// NETWORK 2
// (* End of system generated code, could be modified for your application *)
xExitStop := xCMDwasActive AND NOT stMachineInterface.q_xCmdActive OR xReactionActive;
END_ACTION

ACTION AutoStop_Entry:
(* System generated code, could be modified for your application *)
	xCMDwasActive:=FALSE;
	IF	xReactionActive	THEN
		;
	ELSIF stMachineInterface.q_xCmdDone AND NOT stMachineInterface.q_xCmdActive THEN
		stMachineInterface.iq_diCmd := ET_Cmd.StopAuto;
	ELSE
		stMachineInterface.iq_diCmd := ET_Cmd.Abort;
	END_IF
(* End of system generated code, could be modified for your application *)
END_ACTION

ACTION InitModule_Action:
(* This step is used for initialisations after being enabled *)

(* System generated code, do not change without consulting 'Schneider Electric Automation GmbH' - otherwise you risk instability!!!*)


stMachineInterface.q_xActive		:= TRUE;
stMachineInterface.q_xReady			:= FALSE;
stMachineInterface.q_etDiag			:= GD.ET_Diag.Ok;
stMachineInterface.q_udiDiagExt		:= ET_DiagExt.Initializing;
stMachineInterface.q_sDiagExt		:= FC_EtDiagExtToString(ET_DiagExt.Initializing);
stMachineInterface.q_sMsg			:= '';

stMachineInterface.i_sModuleName		:= 'MainMachine';
stMachineInterface.i_udiModuleId		:= c_udiMainModuleId;
stMachineInterface.i_xLogEnable			:= TRUE;
stMachineInterface.i_wLogDataFilter		:= UDINT_TO_WORD(TPL.ET_LogDataFilter.ModuleDefault);

fbLoggerPoint.RegisterLoggerPoint(	i_ifParent		:= APL.G_ifApplicationLogger,
									i_sName			:= stMachineInterface.i_sModuleName,
									i_sType			:= 'MainMachine',
									i_sSource		:= 'Project',
									q_etDiag		=> ,
									q_etDiagExt		=> );
fbModuleController.RegisterLoggerPoint(	i_ifParent	:= fbLoggerPoint,
										i_sName		:= 'ModuleController',
										q_etDiag	=> ,
										q_etDiagExt	=> );
fbExceptionHandler.RegisterLoggerPoint(	i_ifParent	:= fbLoggerPoint,
										i_sName		:= 'ExceptionHandler',
										q_etDiag	=> ,
										q_etDiagExt	=> );

SYSTEMINTERFACE.FC_DiagNoQuitSet(i_diDiagCode := 8316);
SYSTEMINTERFACE.FC_DiagConfigSet(i_diDiagCode := 8252,i_diDiagClass := 1);
(* End of system generated code, do not change without consulting 'Schneider Electric Automation GmbH' - otherwise you risk instability!!!*)

(* System generated code, could be modified for your application *)
Init_Exceptions();
(* End of system generated code, could be modified for your application *)

(* System generated code, do not change without consulting 'Schneider Electric Automation GmbH' - otherwise you risk instability!!!*)
Init_SubModules();
Init_CmdTables();
Init_Reactions();
UpdateStructs();
(* End of system generated code, do not change without consulting 'Schneider Electric Automation GmbH' - otherwise you risk instability!!!*)

(* System generated code, could be modified for your application *)
Init_Alpha();
Init_Bravo();
Init_MultiCarrier();

xInitSuccessful := TRUE;

(* End of system generated code, could be modified for your application *)

(* Application specific code *)
(* ToDo: Add your application specific code here *)
;
(* End of application specific code *)
END_ACTION

ACTION Input_Action:
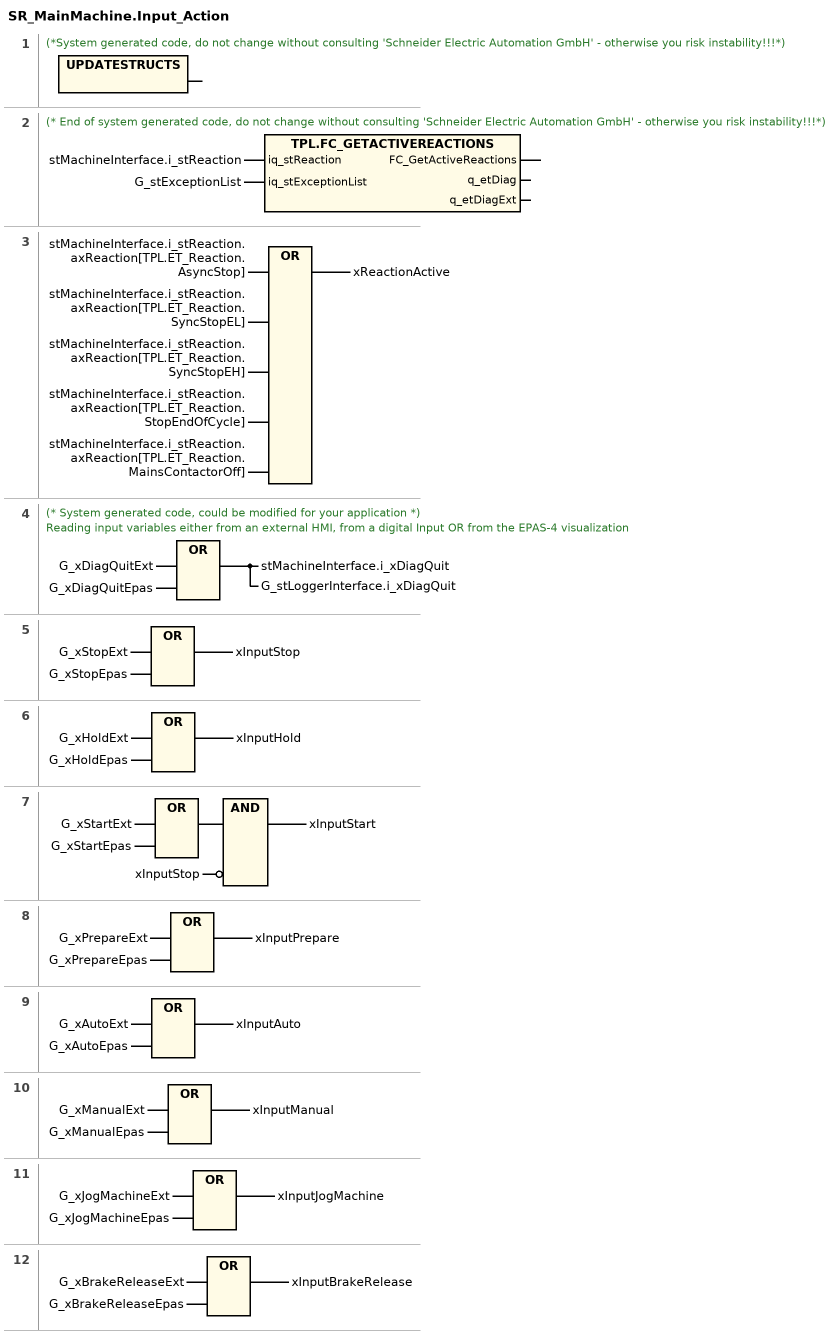
// NETWORK 1
// (*System generated code, do not change without consulting 'Schneider Electric Automation GmbH' - otherwise you risk instability!!!*)
UPDATESTRUCTS();

// NETWORK 2
// (* End of system generated code, do not change without consulting 'Schneider Electric Automation GmbH' - otherwise you risk instability!!!*)
TPL.FC_GETACTIVEREACTIONS(iq_stReaction := stMachineInterface.i_stReaction, iq_stExceptionList := G_stExceptionList);

// NETWORK 3
xReactionActive := stMachineInterface.i_stReaction.axReaction[TPL.ET_Reaction.AsyncStop] OR stMachineInterface.i_stReaction.axReaction[TPL.ET_Reaction.SyncStopEL] OR stMachineInterface.i_stReaction.axReaction[TPL.ET_Reaction.SyncStopEH] OR stMachineInterface.i_stReaction.axReaction[TPL.ET_Reaction.StopEndOfCycle] OR stMachineInterface.i_stReaction.axReaction[TPL.ET_Reaction.MainsContactorOff];

// NETWORK 4
// 					(* System generated code, could be modified for your application *)
// Reading input variables either from an external HMI, from a digital Input OR from the EPAS-4 visualization
//
_w1 := G_xDiagQuitExt OR G_xDiagQuitEpas;
stMachineInterface.i_xDiagQuit := _w1;
G_stLoggerInterface.i_xDiagQuit := _w1;

// NETWORK 5
xInputStop := G_xStopExt OR G_xStopEpas;

// NETWORK 6
xInputHold := G_xHoldExt OR G_xHoldEpas;

// NETWORK 7
xInputStart := (G_xStartExt OR G_xStartEpas) AND NOT xInputStop;

// NETWORK 8
xInputPrepare := G_xPrepareExt OR G_xPrepareEpas;

// NETWORK 9
xInputAuto := G_xAutoExt OR G_xAutoEpas;

// NETWORK 10
xInputManual := G_xManualExt OR G_xManualEpas;

// NETWORK 11
xInputJogMachine := G_xJogMachineExt OR G_xJogMachineEpas;

// NETWORK 12
xInputBrakeRelease := G_xBrakeReleaseExt OR G_xBrakeReleaseEpas;

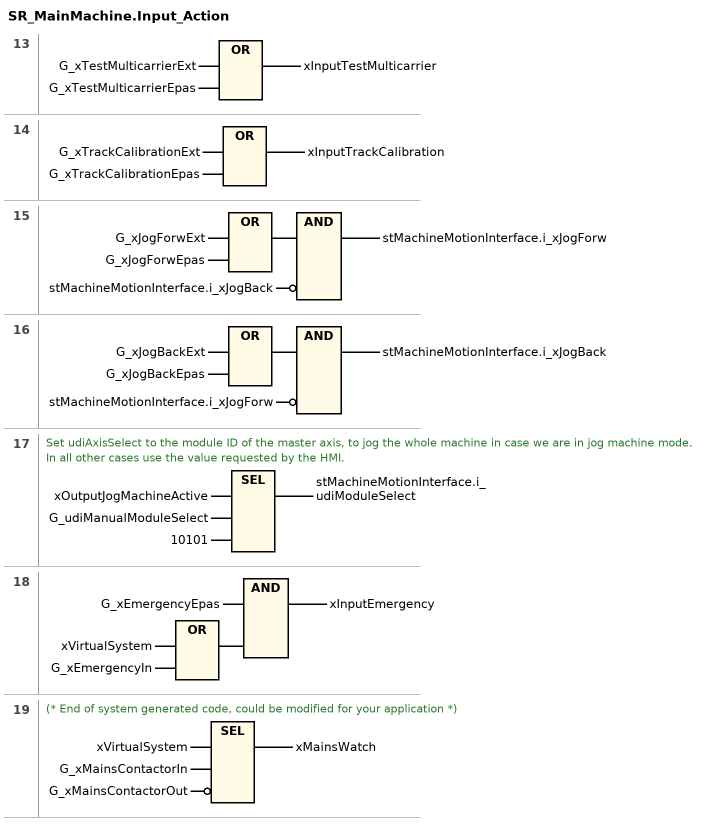
// NETWORK 13
xInputTestMulticarrier := G_xTestMulticarrierExt OR G_xTestMulticarrierEpas;

// NETWORK 14
xInputTrackCalibration := G_xTrackCalibrationExt OR G_xTrackCalibrationEpas;

// NETWORK 15
stMachineMotionInterface.i_xJogForw := (G_xJogForwExt OR G_xJogForwEpas) AND NOT stMachineMotionInterface.i_xJogBack;

// NETWORK 16
stMachineMotionInterface.i_xJogBack := (G_xJogBackExt OR G_xJogBackEpas) AND NOT stMachineMotionInterface.i_xJogForw;

// NETWORK 17
// 					Set udiAxisSelect to the module ID of the master axis, to jog the whole machine in case we are in jog machine mode.
// In all other cases use the value requested by the HMI.
//
stMachineMotionInterface.i_udiModuleSelect := SEL(xOutputJogMachineActive, G_udiManualModuleSelect, 10101);

// NETWORK 18
xInputEmergency := G_xEmergencyEpas AND (xVirtualSystem OR G_xEmergencyIn);

// NETWORK 19
// (* End of system generated code, could be modified for your application *)
xMainsWatch := SEL(xVirtualSystem, G_xMainsContactorIn, NOT G_xMainsContactorOut);
END_ACTION

ACTION JogMachineStep_Action:
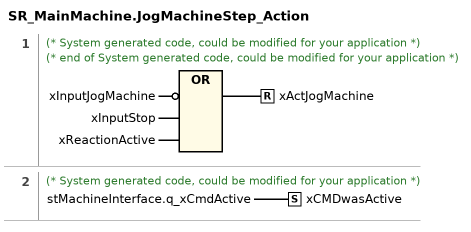
// NETWORK 1
// 					(* System generated code, could be modified for your application *)
// (* end of System generated code, could be modified for your application *)
//
xActJogMachine R= NOT xInputJogMachine OR xInputStop OR xReactionActive;

// NETWORK 2
// (* System generated code, could be modified for your application *)
xCMDwasActive S= stMachineInterface.q_xCmdActive;
END_ACTION

ACTION JogMachineStep_Entry:
(* System generated code, could be modified for your application *)
	xCMDwasActive		:=FALSE;
	stMachineInterface.iq_diCmd	:= ET_Cmd.Jogging;
(* End of system generated code, could be modified for your application *)
END_ACTION

ACTION Logger_Action:
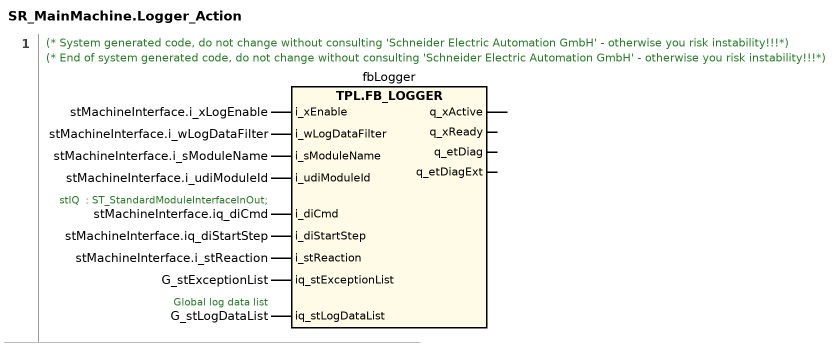
// NETWORK 1
// 					(* System generated code, do not change without consulting 'Schneider Electric Automation GmbH' - otherwise you risk instability!!!*)
// (* End of system generated code, do not change without consulting 'Schneider Electric Automation GmbH' - otherwise you risk instability!!!*)
//
//   fbLogger: Logging related variables
//   stMachineInterface.iq_diCmd: stIQ : ST_StandardModuleInterfaceInOut;
//   G_stLogDataList: Global log data list
fbLogger(
    i_xEnable := stMachineInterface.i_xLogEnable,
    i_wLogDataFilter := stMachineInterface.i_wLogDataFilter,
    i_sModuleName := stMachineInterface.i_sModuleName,
    i_udiModuleId := stMachineInterface.i_udiModuleId,
    i_diCmd := stMachineInterface.iq_diCmd,
    i_diStartStep := stMachineInterface.iq_diStartStep,
    i_stReaction := stMachineInterface.i_stReaction,
    iq_stExceptionList := G_stExceptionList,
    iq_stLogDataList := G_stLogDataList); // TPL.FB_LOGGER
END_ACTION

ACTION ManualStep_Action:
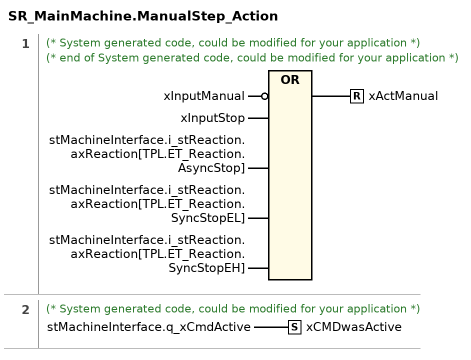
// NETWORK 1
// 					(* System generated code, could be modified for your application *)
// (* end of System generated code, could be modified for your application *)
//
xActManual R= NOT xInputManual OR xInputStop OR stMachineInterface.i_stReaction.axReaction[TPL.ET_Reaction.AsyncStop] OR stMachineInterface.i_stReaction.axReaction[TPL.ET_Reaction.SyncStopEL] OR stMachineInterface.i_stReaction.axReaction[TPL.ET_Reaction.SyncStopEH];

// NETWORK 2
// (* System generated code, could be modified for your application *)
xCMDwasActive S= stMachineInterface.q_xCmdActive;
END_ACTION

ACTION ManualStep_Entry:
(* System generated code, could be modified for your application *)
	xCMDwasActive := FALSE;
	stMachineInterface.iq_diCmd	:= ET_Cmd.Manual;
(* End of system generated code, could be modified for your application *)
END_ACTION

ACTION ModeSelect_Action:
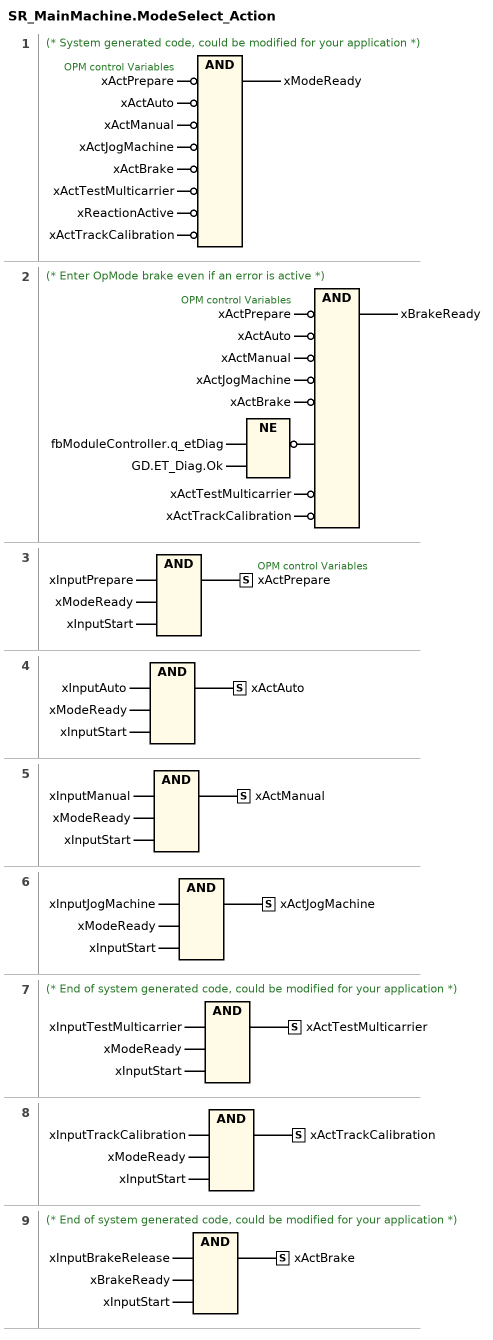
// NETWORK 1
// (* System generated code, could be modified for your application *)
//   xActPrepare: OPM control Variables
xModeReady := NOT xActPrepare AND NOT xActAuto AND NOT xActManual AND NOT xActJogMachine AND NOT xActBrake AND NOT xActTestMulticarrier AND NOT xReactionActive AND NOT xActTrackCalibration;

// NETWORK 2
// (* Enter OpMode brake even if an error is active *)
//   xActPrepare: OPM control Variables
xBrakeReady := NOT xActPrepare AND NOT xActAuto AND NOT xActManual AND NOT xActJogMachine AND NOT xActBrake AND NOT (fbModuleController.q_etDiag <> GD.ET_Diag.Ok) AND NOT xActTestMulticarrier AND NOT xActTrackCalibration;

// NETWORK 3
//   xActPrepare: OPM control Variables
xActPrepare S= xInputPrepare AND xModeReady AND xInputStart;

// NETWORK 4
xActAuto S= xInputAuto AND xModeReady AND xInputStart;

// NETWORK 5
xActManual S= xInputManual AND xModeReady AND xInputStart;

// NETWORK 6
xActJogMachine S= xInputJogMachine AND xModeReady AND xInputStart;

// NETWORK 7
// (* End of system generated code, could be modified for your application *)
xActTestMulticarrier S= xInputTestMulticarrier AND xModeReady AND xInputStart;

// NETWORK 8
xActTrackCalibration S= xInputTrackCalibration AND xModeReady AND xInputStart;

// NETWORK 9
// (* End of system generated code, could be modified for your application *)
xActBrake S= xInputBrakeRelease AND xBrakeReady AND xInputStart;
END_ACTION

ACTION Output_Action:
(* System generated code, could be modified for your application *)
xOutputPrepareActive	:= xActPrepare;
xOutputAutoActive		:= xActAuto;
xOutputManualActive		:= xActManual;
xOutputJogMachineActive	:= xActJogMachine;

IF stMachineInterface.q_udiSubModuleInException <> 0 THEN
	stMachineInterface.q_etDiag		:= GD.ET_Diag.Ok;
	stMachineInterface.q_udiDiagExt	:= ET_DiagExt.SubModuleInException;
	stMachineInterface.q_sDiagExt		:= FC_EtDiagExtToString(ET_DiagExt.SubModuleInException);
	stMachineInterface.q_sMsg			:= '';
ELSE
	IF etDiagModuleController = GD.ET_Diag.Ok THEN
		stMachineInterface.q_etDiag	:= etDiagModuleController;
		stMachineInterface.q_sMsg		:= sMsgModuleController;
		
		CASE etDiagExtModuleController OF
			TPL.ET_DiagExt.DeactivatingSubModules : 
				stMachineInterface.q_udiDiagExt	:= ET_DiagExt.DeactivatingSubModules;
				stMachineInterface.q_sDiagExt		:= FC_EtDiagExtToString(ET_DiagExt.DeactivatingSubModules);
			TPL.ET_DiagExt.Disabled : 
				stMachineInterface.q_udiDiagExt	:= ET_DiagExt.Disabled;
				stMachineInterface.q_sDiagExt		:= FC_EtDiagExtToString(ET_DiagExt.Disabled);
			TPL.ET_DiagExt.ExecuteStep : 
				stMachineInterface.q_udiDiagExt	:= ET_DiagExt.ExecuteStep;
				stMachineInterface.q_sDiagExt		:= FC_EtDiagExtToString(ET_DiagExt.ExecuteStep);
			TPL.ET_DiagExt.Initializing : 
				stMachineInterface.q_udiDiagExt	:= ET_DiagExt.Initializing;
				stMachineInterface.q_sDiagExt		:= FC_EtDiagExtToString(ET_DiagExt.Initializing);
			TPL.ET_DiagExt.WaitAtNegativeStep : 
				stMachineInterface.q_udiDiagExt	:= ET_DiagExt.WaitAtNegativeStep;
				stMachineInterface.q_sDiagExt		:= FC_EtDiagExtToString(ET_DiagExt.WaitAtNegativeStep);
			TPL.ET_DiagExt.WaitCmdsDone : 
				stMachineInterface.q_udiDiagExt	:= ET_DiagExt.WaitCmdsDone;
				stMachineInterface.q_sDiagExt		:= FC_EtDiagExtToString(ET_DiagExt.WaitCmdsDone);
			TPL.ET_DiagExt.WaitForCmd : 
				stMachineInterface.q_udiDiagExt	:= ET_DiagExt.WaitForCmd;
				stMachineInterface.q_sDiagExt		:= FC_EtDiagExtToString(ET_DiagExt.WaitForCmd);
			ELSE
				stMachineInterface.q_etDiag		:= GD. ET_Diag.UnexpectedProgramBehavior;
				stMachineInterface.q_udiDiagExt	:= ET_DiagExt.UnknownStateModuleController;
				stMachineInterface.q_sDiagExt		:= FC_EtDiagExtToString(ET_DiagExt.UnknownStateModuleController);
		END_CASE
	ELSE
		stMachineInterface.q_etDiag		:= GD.ET_Diag.DiagActive;
		stMachineInterface.q_udiDiagExt	:= ET_DiagExt.ModuleControllerException;
		stMachineInterface.q_sDiagExt		:= FC_EtDiagExtToString(ET_DiagExt.ModuleControllerException);
		stMachineInterface.q_sMsg			:= PDL.FC_MultiConcat(	i_sString1 := GD.FC_EtDiagToString(i_etDiag := etDiagModuleController), 
																			i_sString2 := ' - ',
																			i_sString3 := TPL.FC_EtDiagExtToString(etDiagExtModuleController), 
																			i_sString4 := '');
	END_IF
END_IF
(* End of system generated code, only to be changed by experienced programmers *)
END_ACTION

ACTION PrepStep_Action:
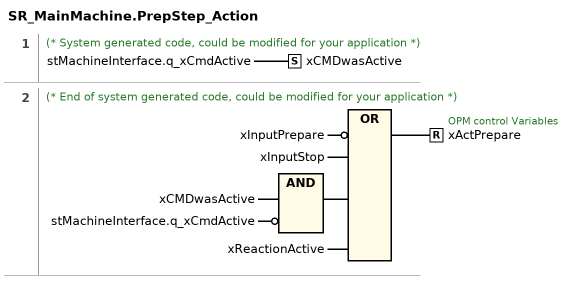
// NETWORK 1
// (* System generated code, could be modified for your application *)
xCMDwasActive S= stMachineInterface.q_xCmdActive;

// NETWORK 2
// (* End of system generated code, could be modified for your application *)
//   xActPrepare: OPM control Variables
xActPrepare R= NOT xInputPrepare OR xInputStop OR xCMDwasActive AND NOT stMachineInterface.q_xCmdActive OR xReactionActive;
END_ACTION

ACTION PrepStep_Entry:
(* System generated code, could be modified for your application *)
	xCMDwasActive:=FALSE;
	stMachineInterface.iq_diCmd	:= ET_Cmd.Prepare;
(* End of system generated code, could be modified for your application *)
END_ACTION

ACTION PrepStop_Action:
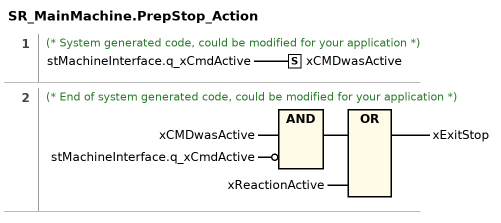
// NETWORK 1
// (* System generated code, could be modified for your application *)
xCMDwasActive S= stMachineInterface.q_xCmdActive;

// NETWORK 2
// (* End of system generated code, could be modified for your application *)
xExitStop := xCMDwasActive AND NOT stMachineInterface.q_xCmdActive OR xReactionActive;
END_ACTION

ACTION PrepStop_Entry:
(* System generated code, could be modified for your application *)
	xCMDwasActive:=FALSE;
	IF	xReactionActive	THEN
		;
	ELSIF stMachineInterface.q_xCmdDone AND NOT stMachineInterface.q_xCmdActive THEN
		stMachineInterface.iq_diCmd	:= ET_Cmd.StopPrepare;
	ELSE
		stMachineInterface.iq_diCmd	:= ET_Cmd.Abort;
	END_IF
(* End of system generated code, could be modified for your application *)
END_ACTION

ACTION Start_Action:
(* This step is active until the machine is being enabled *)	

(* System generated code, do not change without consulting 'Schneider Electric Automation GmbH' - otherwise you risk instability!!!*)
xVirtualSystem := TPL.FC_GetVirtualSystem() AND GVL_Project.Gc_xVirtualMulticarrier;
	
stMachineInterface.q_sModuleTypeName	:= c_sModuleTypeName;
stMachineInterface.q_dwModuleType		:= c_dwModuleType;
stMachineInterface.q_udiModuleVersion	:= c_udiModuleVersion;
(* End of system generated code, do not change without consulting 'Schneider Electric Automation GmbH' - otherwise you risk instability!!!*)

(* System generated code, could be modified for your application *)
IF(SYSTEMINTERFACE.FC_GetPacDriveBootState() <> 1) THEN
	(* avoid starting as long as the boot of the controller is not finished *)
	stMachineInterface.i_xEnable	:= FALSE; (* set transition condition to FALSE ==> ensure that this step stays active *)

	stMachineInterface.q_etDiag		:= GD.ET_Diag.Ok;
	stMachineInterface.q_udiDiagExt	:= ET_DiagExt.WaitUntilControllerFinishedBoot;
	stMachineInterface.q_sDiagExt	:= FC_EtDiagExtToString(stMachineInterface.q_udiDiagExt);
	stMachineInterface.q_sMsg		:= '';
ELSE
	CASE iStateInitMultiCarrier OF
	
	//-------------------------------------------------------------------------------------------------------------------------------------------
	0:  //--- Initialize Hardware interfaces of MultiCarrier devices ---
		stMachineInterface.q_etDiag		:= GD.ET_Diag.Ok;
		stMachineInterface.q_udiDiagExt	:= ET_DiagExt.WaitUntilSercosState4;
		stMachineInterface.q_sDiagExt	:= FC_EtDiagExtToString(stMachineInterface.q_udiDiagExt);
		stMachineInterface.q_sMsg		:= '';
		
		
		
		
		CheckArraySizeOfTrackElements();
		
		IF 	GVL_Project.Gc_xTrackCalibrationOfMulticarrier THEN
			GVL_Project.G_udiUsedNumberOfCarriers := 1;
		ELSE
			GVL_Project.G_udiUsedNumberOfCarriers := GVL_MulticarrierConfiguration.Gc_udiNumberOfCarriers;
		END_IF
		
		IF NOT xError THEN
			SetTrackInterfaces(		q_xError		=> xError,
									q_etDiagExt		=> stMachineInterface.q_udiDiagExt,
									q_sResultMsg	=> stMachineInterface.q_sMsg);
		END_IF
		
		IF NOT xError THEN
			SetSegmentInterfaces(	q_xError		=> xError,
									q_etDiagExt		=> stMachineInterface.q_udiDiagExt,
									q_sResultMsg	=> stMachineInterface.q_sMsg);
		END_IF
								
		IF NOT xError THEN
			SetCarrierInterfaces(	q_xError		=> xError,
									q_etDiagExt		=> stMachineInterface.q_udiDiagExt,
									q_sResultMsg	=> stMachineInterface.q_sMsg);
		END_IF
		
		IF NOT xError THEN
			SetSegmentWorkingMode();
			SetCarrierWorkingMode();	
		END_IF
			
		MC_Track_1.TrackGeometry.Direction	:= GVL_MulticarrierConfiguration.Gc_astTracks[1].xDirection;
		
		IF NOT xError THEN 
			G_ifSercos.PhaseSet := 2;
			iStateInitMultiCarrier := 10;
		ELSE
			iStateInitMultiCarrier 		:= 1000;
		END_IF

	//-------------------------------------------------------------------------------------------------------------------------------------------
	10:	//--- Read Control Loop Parameter
		IF G_ifSercos.State = 2 THEN
			IF NOT GVL_Project.Gc_xVirtualMulticarrier THEN
				SR_ReadControlLoopParameter.ReadParameter();
				iStateInitMultiCarrier := 15;
			ELSE
				iStateInitMultiCarrier := 30;
			END_IF
		END_IF	

	//-------------------------------------------------------------------------------------------------------------------------------------------
	15: //--- Wait for ReadParameterSuccessful
		IF SR_ReadControlLoopParameter.q_xReadParameterDone THEN
			//--- Note on the read parameters:
					//--- After switching on -> the default values are read
					//--- If the system is switched on and only the sercos has been reset, the last written values are read.
			SR_ReadControlLoopParameter.GetParameter(
					q_dwPosP_Straight	=> dwPosP_Straight, 
					q_dwVelP_Straight	=> dwVelP_Straight, 
					q_dwVelI_Straight	=> dwVelI_Straight, 
					q_dwPosP_Curve		=> dwPosP_Curve, 
					q_dwVelP_Curve		=> dwVelP_Curve, 
					q_dwVelI_Curve		=> dwVelI_Curve, 
					q_dwMaxCurr			=> dwMaxCurr, 	 						// Maximum Current in Ampere 				(70 = 1 Ampere )
					q_dwMaxload			=> dwMaxload,   						// load in gramm				    		(Empty Carrier = 800 gramm )
					q_dwDeviationLevelWarning	=> dwDeviationLevelWarning,  	// Warning TrackingDeviation in Increments 	(1600 Increments = 1mm)
					q_dwDeviationLevelError		=> dwDeviationLevelError);	  	// Error TrackingDeviation in Increments 	(1600 Increments = 1mm)
				
			iStateInitMultiCarrier	:= 18;
		ELSIF SR_ReadControlLoopParameter.q_xReadParameterError THEN
			xError								:= TRUE;
			stMachineInterface.q_udiDiagExt  	:= ET_DiagExt.UnexpectedFeedback;
			stMachineInterface.q_sMsg			:= Concat('SR_ReadControlLoopParameter: Result: ' , TO_STRING(SR_ReadControlLoopParameter.diResultSercosReadServiceData) ); 
			iStateInitMultiCarrier 				:= 1000;
		END_IF
		
	//-------------------------------------------------------------------------------------------------------------------------------------------
	18:	//--- Write Control Loop Parameter
		IF G_ifSercos.State = 2 THEN
			IF NOT GVL_Project.Gc_xVirtualMulticarrier THEN
				
				//--- set control loop parameters for trackcalibration
				IF 	GVL_Project.Gc_xTrackCalibrationOfMulticarrier THEN
					dwPosP_Straight := 500;	
					dwVelP_Straight := 2000;
					dwVelI_Straight := 500;
					dwPosP_Curve 	:= 500;	
					dwVelP_Curve 	:= 2000;
					dwVelI_Curve 	:= 500;	
				ELSE
					//-- modify read values if necessary:
					dwPosP_Straight;	
					dwVelP_Straight;
					dwVelI_Straight;
					dwPosP_Curve;
					dwVelP_Curve;
					dwVelI_Curve;
					dwMaxCurr;
					dwMaxload;
					dwDeviationLevelWarning;
					dwDeviationLevelError;
				END_IF
				
				SR_WriteControlLoopParameter.StartAndSetParameter(
												i_dwPosP_Straight 	:= dwPosP_Straight,
												i_dwVelP_Straight 	:= dwVelP_Straight,
												i_dwVelI_Straight 	:= dwVelI_Straight,
												i_dwPosP_Curve 		:= dwPosP_Curve,
												i_dwVelP_Curve 		:= dwVelP_Curve,
												i_dwVelI_Curve 		:= dwVelI_Curve,
												i_dwMaxCurr			:= dwMaxCurr,
												i_dwMaxload			:= dwMaxload,
												i_dwDeviationLevelWarning 	:= dwDeviationLevelWarning,
												i_dwDeviationLevelError 	:= dwDeviationLevelError);		
							
				iStateInitMultiCarrier := 20;
			ELSE
				iStateInitMultiCarrier := 30;
			END_IF
		END_IF	
			
	//-------------------------------------------------------------------------------------------------------------------------------------------
	20: //--- Wait for WriteParameterSuccessful
		IF SR_WriteControlLoopParameter.q_xWriteParameterDone THEN
			iStateInitMultiCarrier	:= 30;
		ELSIF SR_WriteControlLoopParameter.q_xWriteParameterError THEN
			xError								:= TRUE;
			stMachineInterface.q_udiDiagExt  	:= ET_DiagExt.UnexpectedFeedback;
			stMachineInterface.q_sMsg			:= Concat('SR_WriteControlLoopParameter: FC_SercosWriteServiceDataByTopAddr: Result: ' , TO_STRING(SR_WriteControlLoopParameter.diResultSercosWriteServiceData) ); 
			iStateInitMultiCarrier 				:= 1000;
		END_IF
	//-------------------------------------------------------------------------------------------------------------------------------------------
	30:	//--- Set SercosPhase to 4
			CreateTrackForSimulation();
			IF GVL_Project.Gc_xVirtualMulticarrier THEN
				WriteGeometryOnSegments();
			END_IF
			
			
				
			G_ifSercos.PhaseSet 	:= 4;
			iStateInitMultiCarrier	:= 40;
			
	//-------------------------------------------------------------------------------------------------------------------------------------------
	40: //--- Wait Until Sercos State 4
		IF SystemConfiguration.G_ifSercos.State = 4 
		THEN
			stMulticarrierModule.iq_xDoVirtualSetposAfterFirstProgramCall := TRUE;
			
			APL.G_ifApplicationLogger.RegisterCommunicationService(	q_etDiag => ,
																	q_etDiagExt => );	
																	
			stMachineInterface.i_xEnable	:= TRUE;
		END_IF
		
	//-------------------------------------------------------------------------------------------------------------------------------------------
	1000: //--- ErrorState
	//-------------------------------------------------------------------------------------------------------------------------------------------
	
	END_CASE
END_IF
(* End of system generated code, could be modified for your application *)

(* Application specific code *)
(* ToDo: Add your application specific code here *)
;
(* End of application specific code *)
END_ACTION

ACTION StopBrake_Action:
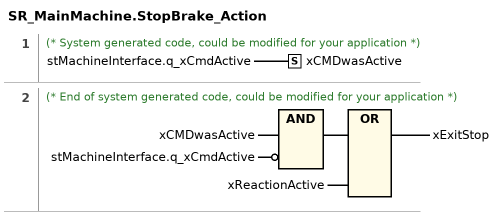
// NETWORK 1
// (* System generated code, could be modified for your application *)
xCMDwasActive S= stMachineInterface.q_xCmdActive;

// NETWORK 2
// (* End of system generated code, could be modified for your application *)
xExitStop := xCMDwasActive AND NOT stMachineInterface.q_xCmdActive OR xReactionActive;
END_ACTION

ACTION StopBrake_Entry:
(* System generated code, could be modified for your application *)
	xCMDwasActive:=FALSE;
	IF	xReactionActive	THEN
		stMachineInterface.iq_diCmd	:= ET_Cmd.Stop;
	ELSIF stMachineInterface.q_xCmdDone AND NOT stMachineInterface.q_xCmdActive THEN
		stMachineInterface.iq_diCmd	:= ET_Cmd.Stop;
	ELSE
		stMachineInterface.iq_diCmd	:= ET_Cmd.Abort;
	END_IF
(* End of system generated code, could be modified for your application *)
END_ACTION

ACTION StopJog_Action:
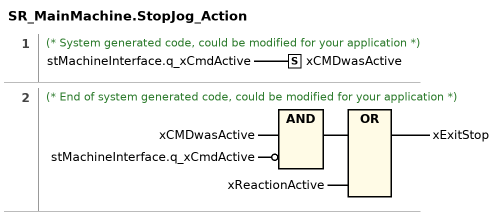
// NETWORK 1
// (* System generated code, could be modified for your application *)
xCMDwasActive S= stMachineInterface.q_xCmdActive;

// NETWORK 2
// (* End of system generated code, could be modified for your application *)
xExitStop := xCMDwasActive AND NOT stMachineInterface.q_xCmdActive OR xReactionActive;
END_ACTION

ACTION StopJog_Entry:
(* System generated code, could be modified for your application *)
	xCMDwasActive:=FALSE;
	IF	xReactionActive	THEN
		;
	ELSIF stMachineInterface.q_xCmdDone AND NOT stMachineInterface.q_xCmdActive THEN
		stMachineInterface.iq_diCmd	:= ET_Cmd.HoldJM;
	ELSE
		stMachineInterface.iq_diCmd	:= ET_Cmd.Abort;
	END_IF
(* End of system generated code, could be modified for your application *)
END_ACTION

ACTION StopMan_Action:
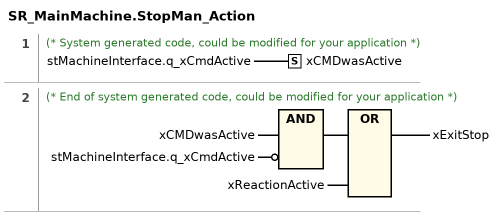
// NETWORK 1
// (* System generated code, could be modified for your application *)
xCMDwasActive S= stMachineInterface.q_xCmdActive;

// NETWORK 2
// (* End of system generated code, could be modified for your application *)
xExitStop := xCMDwasActive AND NOT stMachineInterface.q_xCmdActive OR xReactionActive;
END_ACTION

ACTION StopMan_Entry:
(* System generated code, could be modified for your application *)
	xCMDwasActive:=FALSE;
	IF	xReactionActive	THEN
		;
	ELSIF stMachineInterface.q_xCmdDone AND NOT stMachineInterface.q_xCmdActive THEN
		stMachineInterface.iq_diCmd	:= ET_Cmd.Stop;
	ELSE
		stMachineInterface.iq_diCmd	:= ET_Cmd.Abort;
	END_IF
(* End of system generated code, could be modified for your application *)
END_ACTION

ACTION StopTrackCalibration_Action:
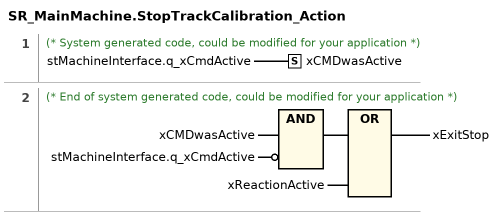
// NETWORK 1
// (* System generated code, could be modified for your application *)
xCMDwasActive S= stMachineInterface.q_xCmdActive;

// NETWORK 2
// (* End of system generated code, could be modified for your application *)
xExitStop := xCMDwasActive AND NOT stMachineInterface.q_xCmdActive OR xReactionActive;
END_ACTION

ACTION StopTrackCalibration_Entry:
(* System generated code, could be modified for your application *)
	xCMDwasActive:=FALSE;
	IF	xReactionActive	THEN
		;
	ELSIF stMachineInterface.q_xCmdDone AND NOT stMachineInterface.q_xCmdActive THEN
		stMachineInterface.iq_diCmd := ET_Cmd.Stop;
	ELSE
		stMachineInterface.iq_diCmd := ET_Cmd.Abort;
	END_IF
(* End of system generated code, could be modified for your application *)
END_ACTION

ACTION SubModules_Action:
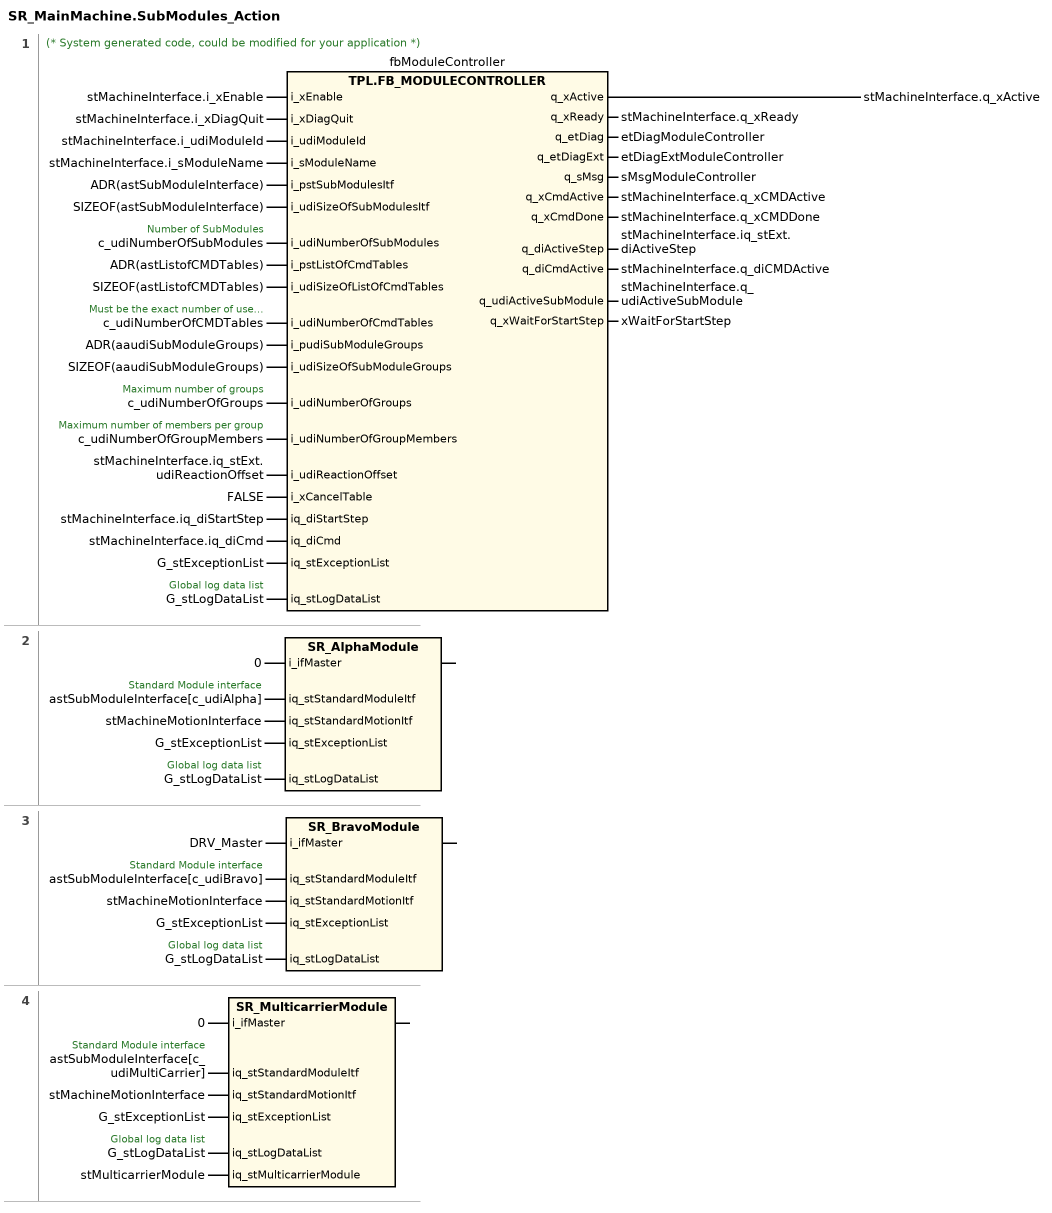
// NETWORK 1
// (* System generated code, could be modified for your application *)
//   fbModuleController: Main ModuleController
//   c_udiNumberOfSubModules: Number of SubModules
//   c_udiNumberOfCMDTables: Must be the exact number of used CMDTables!
//   c_udiNumberOfGroups: Maximum number of groups
//   c_udiNumberOfGroupMembers: Maximum number of members per group
//   G_stLogDataList: Global log data list
fbModuleController(
    i_xEnable := stMachineInterface.i_xEnable,
    i_xDiagQuit := stMachineInterface.i_xDiagQuit,
    i_udiModuleId := stMachineInterface.i_udiModuleId,
    i_sModuleName := stMachineInterface.i_sModuleName,
    i_pstSubModulesItf := ADR(astSubModuleInterface),
    i_udiSizeOfSubModulesItf := SIZEOF(astSubModuleInterface),
    i_udiNumberOfSubModules := c_udiNumberOfSubModules,
    i_pstListOfCmdTables := ADR(astListofCMDTables),
    i_udiSizeOfListOfCmdTables := SIZEOF(astListofCMDTables),
    i_udiNumberOfCmdTables := c_udiNumberOfCMDTables,
    i_pudiSubModuleGroups := ADR(aaudiSubModuleGroups),
    i_udiSizeOfSubModuleGroups := SIZEOF(aaudiSubModuleGroups),
    i_udiNumberOfGroups := c_udiNumberOfGroups,
    i_udiNumberOfGroupMembers := c_udiNumberOfGroupMembers,
    i_udiReactionOffset := stMachineInterface.iq_stExt.udiReactionOffset,
    i_xCancelTable := FALSE,
    iq_diStartStep := stMachineInterface.iq_diStartStep,
    iq_diCmd := stMachineInterface.iq_diCmd,
    iq_stExceptionList := G_stExceptionList,
    iq_stLogDataList := G_stLogDataList,
    q_xReady => stMachineInterface.q_xReady,
    q_etDiag => etDiagModuleController,
    q_etDiagExt => etDiagExtModuleController,
    q_sMsg => sMsgModuleController,
    q_xCmdActive => stMachineInterface.q_xCMDActive,
    q_xCmdDone => stMachineInterface.q_xCMDDone,
    q_diActiveStep => stMachineInterface.iq_stExt.diActiveStep,
    q_diCmdActive => stMachineInterface.q_diCMDActive,
    q_udiActiveSubModule => stMachineInterface.q_udiActiveSubModule,
    q_xWaitForStartStep => xWaitForStartStep); // TPL.FB_MODULECONTROLLER
stMachineInterface.q_xActive := fbModuleController.q_xActive;

// NETWORK 2
//   astSubModuleInterface[c_udiAlpha]: Standard Module interface
//   G_stLogDataList: Global log data list
SR_AlphaModule(i_ifMaster := 0, iq_stStandardModuleItf := astSubModuleInterface[c_udiAlpha], iq_stStandardMotionItf := stMachineMotionInterface, iq_stExceptionList := G_stExceptionList, iq_stLogDataList := G_stLogDataList);

// NETWORK 3
//   astSubModuleInterface[c_udiBravo]: Standard Module interface
//   G_stLogDataList: Global log data list
SR_BravoModule(i_ifMaster := DRV_Master, iq_stStandardModuleItf := astSubModuleInterface[c_udiBravo], iq_stStandardMotionItf := stMachineMotionInterface, iq_stExceptionList := G_stExceptionList, iq_stLogDataList := G_stLogDataList);

// NETWORK 4
//   astSubModuleInterface[c_udiMultiCarrier]: Standard Module interface
//   G_stLogDataList: Global log data list
SR_MulticarrierModule(i_ifMaster := 0, iq_stStandardModuleItf := astSubModuleInterface[c_udiMultiCarrier], iq_stStandardMotionItf := stMachineMotionInterface, iq_stExceptionList := G_stExceptionList, iq_stLogDataList := G_stLogDataList, iq_stMulticarrierModule := stMulticarrierModule);
END_ACTION

ACTION TestMulticarrierStep_Action:
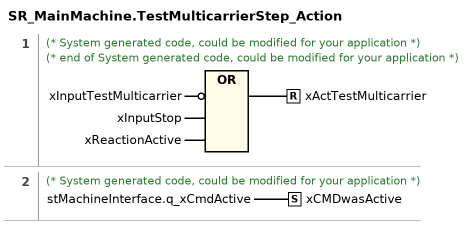
// NETWORK 1
// 					(* System generated code, could be modified for your application *)
// (* end of System generated code, could be modified for your application *)
//
xActTestMulticarrier R= NOT xInputTestMulticarrier OR xInputStop OR xReactionActive;

// NETWORK 2
// (* System generated code, could be modified for your application *)
xCMDwasActive S= stMachineInterface.q_xCmdActive;
END_ACTION

ACTION TestMulticarrierStep_Entry:
(* System generated code, could be modified for your application *)
	xCmdWasActive := FALSE;
	stMachineInterface.iq_diCmd := ET_Cmd.TestMulticarrier;
(* End of system generated code, could be modified for your application *)
END_ACTION

ACTION TestMulticarrierStop_Action:
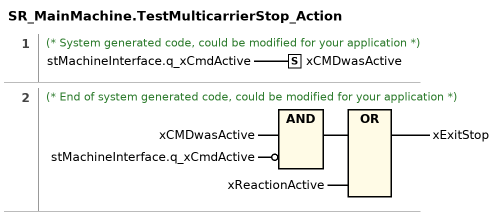
// NETWORK 1
// (* System generated code, could be modified for your application *)
xCMDwasActive S= stMachineInterface.q_xCmdActive;

// NETWORK 2
// (* End of system generated code, could be modified for your application *)
xExitStop := xCMDwasActive AND NOT stMachineInterface.q_xCmdActive OR xReactionActive;
END_ACTION

ACTION TestMulticarrierStop_Entry:
(* System generated code, could be modified for your application *)
	xCMDwasActive:=FALSE;
	IF	xReactionActive	THEN
		;
	ELSIF stMachineInterface.q_xCmdDone AND NOT stMachineInterface.q_xCmdActive THEN
		stMachineInterface.iq_diCmd := ET_Cmd.Stop;
	ELSE
		stMachineInterface.iq_diCmd := ET_Cmd.Abort;
	END_IF
(* End of system generated code, could be modified for your application *)
END_ACTION

ACTION TrackCalibrationStep_Action:
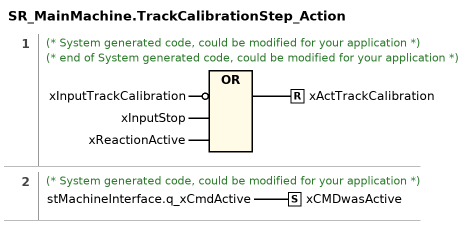
// NETWORK 1
// 					(* System generated code, could be modified for your application *)
// (* end of System generated code, could be modified for your application *)
//
xActTrackCalibration R= NOT xInputTrackCalibration OR xInputStop OR xReactionActive;

// NETWORK 2
// (* System generated code, could be modified for your application *)
xCMDwasActive S= stMachineInterface.q_xCmdActive;
END_ACTION

ACTION TrackCalibrationStep_Entry:
(* System generated code, could be modified for your application *)
	xCmdWasActive := FALSE;
	stMachineInterface.iq_diCmd := ET_Cmd.TrackCalibration;
(* End of system generated code, could be modified for your application *)
END_ACTION

ACTION UpdateStructs:
(* System generated code, do not change without consulting 'Schneider Electric Automation GmbH' - otherwise you risk instability!!!*)
fbDetectOnlineChange(	i_xEnable	:= TRUE, 
						i_xDetect	:= TRUE, 
						q_xActive	=> xDetectOnlineChangeActive, 
						q_xReady	=> xDetectOnlineChangeReady, 
						q_etDiag	=> etDetectOnlineChangeDiag, 
						q_etDiagExt	=> etDetectOnlineChangeDiagExt, 
						q_sMsg		=> sDetectOnlineChangeMsg, 
						q_xChange	=> );
						
IF(NOT fbDetectOnlineChange.q_xChange) THEN
	RETURN;
END_IF

stMachineInterface.iq_stExt.udiNumberOfSubModules 		:= c_udiNumberOfSubModules;
stMachineInterface.iq_stExt.dwSubModulesItf		 		:= ADR(astSubModuleInterface);
stMachineInterface.iq_stExt.pdwSubModulesAddItf			:= ADR(adwSubModuleAddInterfaces);
stMachineInterface.iq_stExt.pstListofCMDTables			:= ADR(astListOfCMDTables);
stMachineInterface.iq_stExt.udiNumberOfCmdTables		:= c_udiNumberOfCMDTables;
(* End of system generated code, do not change without consulting 'Schneider Electric Automation GmbH' - otherwise you risk instability!!!*)

(* System generated code, could be modified for your application *)

xUpdateStructsException := FALSE;

//-------------------------------------------------------------------------------------------------------------------
//-- Update CmdTable - Prepare 
	//
	TPL.FC_UpdateCmdTableListElement(	i_pstListofCMDTables	:= ADR(astListofCMDTables),
										i_udiNumberOfCmdTables	:= c_udiNumberOfCMDTables,
										i_diCMD					:= ET_Cmd.Prepare,
										i_pstCMDTable			:= ADR(astPrepareTable),
										q_etDiag				=> etDiag,
										q_etDiagExt				=> etDiagExtTPL);
										
	IF etDiag <> GD.ET_Diag.Ok AND NOT xUpdateStructsException THEN
		xUpdateStructsException := TRUE;
		
		stUpdateStructsException.sMsg := PDL.FC_MultiConcat(i_sString1 := 'Update CmdTable: Prepare - ', 
															i_sString2 := GD.FC_EtDiagToString(i_etDiag := etDiag), 
															i_sString3 := ' - ', 
															i_sString4 := TPL.FC_EtDiagExtToString(i_etDiagExt := etDiagExtTPL));
	END_IF										

//-------------------------------------------------------------------------------------------------------------------
//-- Update CmdTable - Auto 
	//
	TPL.FC_UpdateCmdTableListElement(	i_pstListofCMDTables	:= ADR(astListofCMDTables),
										i_udiNumberOfCMDTables	:= c_udiNumberOfCMDTables,
										i_diCMD					:= ET_Cmd.Auto,
										i_pstCMDTable			:= ADR(astAutoTable),
										q_etDiag				=> etDiag,
										q_etDiagExt				=> etDiagExtTPL);
										
	IF etDiag <> GD.ET_Diag.Ok AND NOT xUpdateStructsException THEN
		xUpdateStructsException := TRUE;
		
		stUpdateStructsException.sMsg := PDL.FC_MultiConcat(i_sString1 := 'Update CmdTable: Auto - ', 
															i_sString2 := GD.FC_EtDiagToString(i_etDiag := etDiag), 
															i_sString3 := ' - ', 
															i_sString4 := TPL.FC_EtDiagExtToString(i_etDiagExt := etDiagExtTPL));
	END_IF		

//-------------------------------------------------------------------------------------------------------------------
//-- Update CmdTable - Manual 
	//
	TPL.FC_UpdateCmdTableListElement(	i_pstListofCMDTables	:= ADR(astListofCMDTables),
										i_udiNumberOfCMDTables	:= c_udiNumberOfCMDTables,
										i_diCMD					:= ET_Cmd.Manual,
										i_pstCMDTable			:= ADR(astManualTable),
										q_etDiag				=> etDiag,
										q_etDiagExt				=> etDiagExtTPL);
										
	IF etDiag <> GD.ET_Diag.Ok AND NOT xUpdateStructsException THEN
		xUpdateStructsException := TRUE;
		
		stUpdateStructsException.sMsg := PDL.FC_MultiConcat(i_sString1 := 'Update CmdTable: Manual - ', 
															i_sString2 := GD.FC_EtDiagToString(i_etDiag := etDiag), 
															i_sString3 := ' - ', 
															i_sString4 := TPL.FC_EtDiagExtToString(i_etDiagExt := etDiagExtTPL));
	END_IF		

//-------------------------------------------------------------------------------------------------------------------
//-- Update CmdTable - Stop 
	//
	TPL.FC_UpdateCmdTableListElement(	i_pstListofCMDTables	:= ADR(astListofCMDTables),
										i_udiNumberOfCMDTables	:= c_udiNumberOfCMDTables,
										i_diCMD					:= ET_Cmd.Stop,
										i_pstCMDTable			:= ADR(astStopTable),
										q_etDiag				=> etDiag,
										q_etDiagExt				=> etDiagExtTPL);
										
	IF etDiag <> GD.ET_Diag.Ok AND NOT xUpdateStructsException THEN
		xUpdateStructsException := TRUE;
		
		stUpdateStructsException.sMsg := PDL.FC_MultiConcat(i_sString1 := 'Update CmdTable: Stop - ', 
															i_sString2 := GD.FC_EtDiagToString(i_etDiag := etDiag), 
															i_sString3 := ' - ', 
															i_sString4 := TPL.FC_EtDiagExtToString(i_etDiagExt := etDiagExtTPL));
	END_IF		

//-------------------------------------------------------------------------------------------------------------------
//-- Update CmdTable - Start 
	//
	TPL.FC_UpdateCmdTableListElement(	i_pstListofCMDTables	:= ADR(astListofCMDTables),
										i_udiNumberOfCMDTables	:= c_udiNumberOfCMDTables,
										i_diCMD					:= ET_Cmd.Start,
										i_pstCMDTable			:= ADR(astStartTable),
										q_etDiag				=> etDiag,
										q_etDiagExt				=> etDiagExtTPL);
										
	IF etDiag <> GD.ET_Diag.Ok AND NOT xUpdateStructsException THEN
		xUpdateStructsException := TRUE;
		
		stUpdateStructsException.sMsg := PDL.FC_MultiConcat(i_sString1 := 'Update CmdTable: Start - ', 
															i_sString2 := GD.FC_EtDiagToString(i_etDiag := etDiag), 
															i_sString3 := ' - ', 
															i_sString4 := TPL.FC_EtDiagExtToString(i_etDiagExt := etDiagExtTPL));
	END_IF		

//-------------------------------------------------------------------------------------------------------------------
//-- Update CmdTable - Abort 
	//
	TPL.FC_UpdateCmdTableListElement(	i_pstListofCMDTables	:= ADR(astListofCMDTables),
										i_udiNumberOfCMDTables	:= c_udiNumberOfCMDTables,
										i_diCMD					:= ET_Cmd.Abort,
										i_pstCMDTable			:= ADR(astAbortTable),
										q_etDiag				=> etDiag,
										q_etDiagExt				=> etDiagExtTPL);
										
	IF etDiag <> GD.ET_Diag.Ok AND NOT xUpdateStructsException THEN
		xUpdateStructsException := TRUE;
		
		stUpdateStructsException.sMsg := PDL.FC_MultiConcat(i_sString1 := 'Update CmdTable: Abort - ', 
															i_sString2 := GD.FC_EtDiagToString(i_etDiag := etDiag), 
															i_sString3 := ' - ', 
															i_sString4 := TPL.FC_EtDiagExtToString(i_etDiagExt := etDiagExtTPL));
	END_IF		

//-------------------------------------------------------------------------------------------------------------------
//-- Update CmdTable - Hold 
	//
	TPL.FC_UpdateCmdTableListElement(	i_pstListofCMDTables	:= ADR(astListofCMDTables),
										i_udiNumberOfCMDTables	:= c_udiNumberOfCMDTables,
										i_diCMD					:= ET_Cmd.Hold,
										i_pstCMDTable			:= ADR(astHoldTable),
										q_etDiag				=> etDiag,
										q_etDiagExt				=> etDiagExtTPL);
										
	IF etDiag <> GD.ET_Diag.Ok AND NOT xUpdateStructsException THEN
		xUpdateStructsException := TRUE;
		
		stUpdateStructsException.sMsg := PDL.FC_MultiConcat(i_sString1 := 'Update CmdTable: Hold - ', 
															i_sString2 := GD.FC_EtDiagToString(i_etDiag := etDiag), 
															i_sString3 := ' - ', 
															i_sString4 := TPL.FC_EtDiagExtToString(i_etDiagExt := etDiagExtTPL));
	END_IF		

//-------------------------------------------------------------------------------------------------------------------
//-- Update CmdTable - BrakeRelease 
	//
	TPL.FC_UpdateCmdTableListElement(	i_pstListofCMDTables	:= ADR(astListofCMDTables),
										i_udiNumberOfCMDTables	:= c_udiNumberOfCMDTables,
										i_diCMD					:= ET_Cmd.HoldJM,
										i_pstCMDTable			:= ADR(astHoldJogMachineTable),
										q_etDiag				=> etDiag,
										q_etDiagExt				=> etDiagExtTPL);
										
	IF etDiag <> GD.ET_Diag.Ok AND NOT xUpdateStructsException THEN
		xUpdateStructsException := TRUE;
		
		stUpdateStructsException.sMsg := PDL.FC_MultiConcat(i_sString1 := 'Update CmdTable: HoldJogMachine - ', 
															i_sString2 := GD.FC_EtDiagToString(i_etDiag := etDiag), 
															i_sString3 := ' - ', 
															i_sString4 := TPL.FC_EtDiagExtToString(i_etDiagExt := etDiagExtTPL));
	END_IF		
//-------------------------------------------------------------------------------------------------------------------
//-- Update CmdTable - TestMulticarrier 
	//
	TPL.FC_UpdateCmdTableListElement(	i_pstListofCMDTables	:= ADR(astListofCMDTables),
										i_udiNumberOfCMDTables	:= c_udiNumberOfCMDTables,
										i_diCMD					:= ET_Cmd.TestMulticarrier,
										i_pstCMDTable			:= ADR(astTestMulticarrierTable),
										q_etDiag				=> etDiag,
										q_etDiagExt				=> etDiagExtTPL);
										
	IF etDiag <> GD.ET_Diag.Ok AND NOT xUpdateStructsException THEN
		xUpdateStructsException := TRUE;
		
		stUpdateStructsException.sMsg := PDL.FC_MultiConcat(i_sString1 := 'Update CmdTable: TestMulticarrier - ', 
															i_sString2 := GD.FC_EtDiagToString(i_etDiag := etDiag), 
															i_sString3 := ' - ', 
															i_sString4 := TPL.FC_EtDiagExtToString(i_etDiagExt := etDiagExtTPL));
	END_IF		
//-------------------------------------------------------------------------------------------------------------------
//-- Update CmdTable - TrackCalibration 
	//
	TPL.FC_UpdateCmdTableListElement(	i_pstListofCMDTables	:= ADR(astListofCMDTables),
										i_udiNumberOfCMDTables	:= c_udiNumberOfCMDTables,
										i_diCMD					:= ET_Cmd.TrackCalibration,
										i_pstCMDTable			:= ADR(astTrackCalibrationTable),
										q_etDiag				=> etDiag,
										q_etDiagExt				=> etDiagExtTPL);
										
	IF etDiag <> GD.ET_Diag.Ok AND NOT xUpdateStructsException THEN
		xUpdateStructsException := TRUE;
		
		stUpdateStructsException.sMsg := PDL.FC_MultiConcat(i_sString1 := 'Update CmdTable: TrackCalibration - ', 
															i_sString2 := GD.FC_EtDiagToString(i_etDiag := etDiag), 
															i_sString3 := ' - ', 
															i_sString4 := TPL.FC_EtDiagExtToString(i_etDiagExt := etDiagExtTPL));
	END_IF		
//-------------------------------------------------------------------------------------------------------------------
//-- Update CmdTable - StopPrepare 
	//
	TPL.FC_UpdateCmdTableListElement(	i_pstListofCMDTables	:= ADR(astListofCMDTables),
										i_udiNumberOfCMDTables	:= c_udiNumberOfCMDTables,
										i_diCMD					:= ET_Cmd.StopPrepare,
										i_pstCMDTable			:= ADR(astStopPrepareTable),
										q_etDiag				=> etDiag,
										q_etDiagExt				=> etDiagExtTPL);
										
	IF etDiag <> GD.ET_Diag.Ok AND NOT xUpdateStructsException THEN
		xUpdateStructsException := TRUE;
		
		stUpdateStructsException.sMsg := PDL.FC_MultiConcat(i_sString1 := 'Update CmdTable: StopPrepare - ', 
															i_sString2 := GD.FC_EtDiagToString(i_etDiag := etDiag), 
															i_sString3 := ' - ', 
															i_sString4 := TPL.FC_EtDiagExtToString(i_etDiagExt := etDiagExtTPL));
	END_IF	
//-------------------------------------------------------------------------------------------------------------------
//-- Update CmdTable - StopAuto 
	//
	TPL.FC_UpdateCmdTableListElement(	i_pstListofCMDTables	:= ADR(astListofCMDTables),
										i_udiNumberOfCMDTables	:= c_udiNumberOfCMDTables,
										i_diCMD					:= ET_Cmd.StopAuto,
										i_pstCMDTable			:= ADR(astStopAutoTable),
										q_etDiag				=> etDiag,
										q_etDiagExt				=> etDiagExtTPL);
										
	IF etDiag <> GD.ET_Diag.Ok AND NOT xUpdateStructsException THEN
		xUpdateStructsException := TRUE;
		
		stUpdateStructsException.sMsg := PDL.FC_MultiConcat(i_sString1 := 'Update CmdTable: StopAuto - ', 
															i_sString2 := GD.FC_EtDiagToString(i_etDiag := etDiag), 
															i_sString3 := ' - ', 
															i_sString4 := TPL.FC_EtDiagExtToString(i_etDiagExt := etDiagExtTPL));
	END_IF	
	
	
//-------------------------------------------------------------------------------------------------------------------
//-- Update AddInterface - BrakeRelease 
	//
	TPL.FC_UpdateCmdTableListElement(	i_pstListofCMDTables	:= ADR(astListofCMDTables),
										i_udiNumberOfCMDTables	:= c_udiNumberOfCMDTables,
										i_diCMD					:= ET_Cmd.BrakeRelease,
										i_pstCMDTable			:= ADR(astBrakeReleaseTable),
										q_etDiag				=> etDiag,
										q_etDiagExt				=> etDiagExtTPL);
										
	IF etDiag <> GD.ET_Diag.Ok AND NOT xUpdateStructsException THEN
		xUpdateStructsException := TRUE;
		
		stUpdateStructsException.sMsg := PDL.FC_MultiConcat(i_sString1 := 'Update CmdTable: BrakeRelease - ', 
															i_sString2 := GD.FC_EtDiagToString(i_etDiag := etDiag), 
															i_sString3 := ' - ', 
															i_sString4 := TPL.FC_EtDiagExtToString(i_etDiagExt := etDiagExtTPL));
	END_IF		
									
//-------------------------------------------------------------------------------------------------------------------
//-- Update AddInterface - Jogging 
	//
	TPL.FC_UpdateCmdTableListElement(	i_pstListofCMDTables	:= ADR(astListofCMDTables),
										i_udiNumberOfCMDTables	:= c_udiNumberOfCMDTables,
										i_diCMD					:= ET_Cmd.Jogging,
										i_pstCMDTable			:= ADR(astJogMachineTable),
										q_etDiag				=> etDiag,
										q_etDiagExt				=> etDiagExtTPL);
										
	IF etDiag <> GD.ET_Diag.Ok AND NOT xUpdateStructsException THEN
		xUpdateStructsException := TRUE;
		
		stUpdateStructsException.sMsg := PDL.FC_MultiConcat(i_sString1 := 'Update CmdTable: Jogging - ', 
															i_sString2 := GD.FC_EtDiagToString(i_etDiag := etDiag), 
															i_sString3 := ' - ', 
															i_sString4 := TPL.FC_EtDiagExtToString(i_etDiagExt := etDiagExtTPL));
	END_IF		
//-------------------------------------------------------------------------------------------------------------------
//-- Update AddInterface - Alpha 
	//
	TPL.FC_UpdateNodeModuleAddInterfaceStruct(	i_pdwSubModulesAddItf		:= ADR(adwSubModuleAddInterfaces),
												i_udiSubModuleConstant		:= c_udiAlpha,
												q_etDiag					=> etDiag,
												q_etDiagExt					=> etDiagExtTPL);
										
	IF etDiag <> GD.ET_Diag.Ok AND NOT xUpdateStructsException THEN
		xUpdateStructsException := TRUE;
		
		stUpdateStructsException.sMsg := PDL.FC_MultiConcat(i_sString1 := 'Update AddInterface: Alpha - ', 
															i_sString2 := GD.FC_EtDiagToString(i_etDiag := etDiag), 
															i_sString3 := ' - ', 
															i_sString4 := TPL.FC_EtDiagExtToString(i_etDiagExt := etDiagExtTPL));
	END_IF		
									
//-------------------------------------------------------------------------------------------------------------------
//-- Update AddInterface - Bravo 
	//
	TPL.FC_UpdateNodeModuleAddInterfaceStruct(	i_pdwSubModulesAddItf		:= ADR(adwSubModuleAddInterfaces),
												i_udiSubModuleConstant		:= c_udiBravo,
												q_etDiag					=> etDiag,
												q_etDiagExt					=> etDiagExtTPL);
										
	IF etDiag <> GD.ET_Diag.Ok AND NOT xUpdateStructsException THEN
		xUpdateStructsException := TRUE;
		
		stUpdateStructsException.sMsg := PDL.FC_MultiConcat(i_sString1 := 'Update AddInterface: Bravo - ', 
															i_sString2 := GD.FC_EtDiagToString(i_etDiag := etDiag), 
															i_sString3 := ' - ', 
															i_sString4 := TPL.FC_EtDiagExtToString(i_etDiagExt := etDiagExtTPL));
	END_IF		
									
//-------------------------------------------------------------------------------------------------------------------
//-- Update AddInterface - MultiCarrier 
	//
	TPL.FC_UpdateNodeModuleAddInterfaceStruct(	i_pdwSubModulesAddItf		:= ADR(adwSubModuleAddInterfaces),
												i_udiSubModuleConstant		:= c_udiMultiCarrier,
												q_etDiag					=> etDiag,
												q_etDiagExt					=> etDiagExtTPL);
										
	IF etDiag <> GD.ET_Diag.Ok AND NOT xUpdateStructsException THEN
		xUpdateStructsException := TRUE;
		
		stUpdateStructsException.sMsg := PDL.FC_MultiConcat(i_sString1 := 'Update AddInterface: MultiCarrier - ', 
															i_sString2 := GD.FC_EtDiagToString(i_etDiag := etDiag), 
															i_sString3 := ' - ', 
															i_sString4 := TPL.FC_EtDiagExtToString(i_etDiagExt := etDiagExtTPL));
	END_IF		

//-------------------------------------------------------------------------------------------------------------------
//-- Set exception if any exception occurred *)
	//
	fbExceptionHandler.SetException(i_xExceptionActive	:= xUpdateStructsException, 
									iq_stException		:= stUpdateStructsException, 
									iq_stExceptionList	:= G_stExceptionList);
						
	xInitSuccessful := xInitSuccessful AND NOT xUpdateStructsException;
	
	etDiag := GD.ET_Diag.Ok;

(* End of system generated code, could be modified for your application *)
END_ACTION

END_PROGRAM

// LMC_PacDrive/Application/TemplateFullProgrammingFramework/ProjectDiagnostics/FC_EtDiagExtToString
FUNCTION FC_EtDiagExtToString : STRING[80]
VAR_INPUT
	i_etDiagExt : ET_DiagExt;
END_VAR
VAR_OUTPUT
	q_etDiag	: GD.ET_Diag := GD.ET_Diag.Ok;
	q_etDiagExt	: ET_DiagExt := ET_DiagExt.Ok;
END_VAR

CASE i_etDiagExt OF
	ET_DiagExt.Ok:								FC_EtDiagExtToString := 'Ok';
	ET_DiagExt.Disabled:						FC_EtDiagExtToString := 'Disabled';
	ET_DiagExt.WaitUntilControllerFinishedBoot:	FC_EtDiagExtToString := 'WaitUntilControllerFinishedBoot';
	ET_DiagExt.Initializing:					FC_EtDiagExtToString := 'Initializing';
	ET_DiagExt.DeactivatingSubModules:			FC_EtDiagExtToString := 'DeactivatingSubModules';
	ET_DiagExt.ExecuteStep:						FC_EtDiagExtToString := 'ExecuteStep';
	ET_DiagExt.WaitAtNegativeStep:				FC_EtDiagExtToString := 'WaitAtNegativeStep';
	ET_DiagExt.WaitCmdsDone:					FC_EtDiagExtToString := 'WaitCmdsDone';
	ET_DiagExt.WaitForCmd:						FC_EtDiagExtToString := 'WaitForCmd';
	ET_DiagExt.SubModuleInException:			FC_EtDiagExtToString := 'SubModuleInException';
	ET_DiagExt.ModuleControllerException:		FC_EtDiagExtToString := 'ModuleControllerException';
	ET_DiagExt.UnknownStateModuleController:	FC_EtDiagExtToString := 'UnknownStateModuleController';
	
	ET_DiagExt.SystemFatalException:			FC_EtDiagExtToString := 'SystemFatalException';
	ET_DiagExt.SystemException:					FC_EtDiagExtToString := 'SystemException';
	ET_DiagExt.SystemWarning:					FC_EtDiagExtToString := 'SystemWarning';
	ET_DiagExt.MainSystemEmergencyStop:			FC_EtDiagExtToString := 'MainSystemEmergencyStop';
	ET_DiagExt.InvalidPointer:					FC_EtDiagExtToString := 'InvalidPointer';
	ET_DiagExt.UpdateStructsException:			FC_EtDiagExtToString := 'UpdateStructsException';
	ET_DiagExt.InitReactionsException:			FC_EtDiagExtToString := 'InitReactionsException';
	ET_DiagExt.InitSubModulesException:			FC_EtDiagExtToString := 'InitSubModulesException';
	ET_DiagExt.ifMulticarrierSegmentsInvalid :					FC_EtDiagExtToString := 'ifMulticarrierSegmentsInvalid ';
	ET_DiagExt.UnknownDiagExt:					FC_EtDiagExtToString := 'UnknownDiagExt';

	ET_DiagExt.Exception1FromVis:				FC_EtDiagExtToString := 'Exception1FromVis';
	ET_DiagExt.Exception2FromVis:				FC_EtDiagExtToString := 'Exception2FromVis';
	ET_DiagExt.Exception3FromVis:				FC_EtDiagExtToString := 'Exception3FromVis';
	ET_DiagExt.Exception4FromVis:				FC_EtDiagExtToString := 'Exception4FromVis';
	ET_DiagExt.Exception5FromVis:				FC_EtDiagExtToString := 'Exception5FromVis';
	
	ET_DiagExt.DiagnosticsWarning:				FC_EtDiagExtToString := 'DiagnosticsWarning';
	ET_DiagExt.WaitUntilDiagnosticsManagerReady:FC_EtDiagExtToString := 'WaitUntilDiagnosticsManagerReady';
	ET_DiagExt.WaitUntilDisabled:				FC_EtDiagExtToString := 'WaitUntilDisabled';
	ET_DiagExt.WaitUntilDiagSourceRegistered:	FC_EtDiagExtToString := 'WaitUntilDiagSourceRegistered';
	ET_DiagExt.WaitForCommunication:			FC_EtDiagExtToString := 'WaitForCommunication';
	ET_DiagExt.DataSuccessfullyWritten:			FC_EtDiagExtToString := 'DataSuccessfullyWritten';
	ET_DiagExt.WritingToFile:					FC_EtDiagExtToString := 'WritingToFile';
	ET_DiagExt.FileIdInvalid:					FC_EtDiagExtToString := 'FileIdInvalid';
	ET_DiagExt.CmdUnknown:						FC_EtDiagExtToString := 'CmdUnknown';
	ET_DiagExt.WaitUntilSercosState4:			FC_EtDiagExtToString := 'WaitUntilSercosState4';
	ET_DiagExt.UnexpectedFeedback:				FC_EtDiagExtToString := 'UnexpectedFeedback';
	ET_DiagExt.UnknownDiagExtUser:				FC_EtDiagExtToString := 'UnknownDiagExtUser';
	ET_DiagExt.HardwareException:				FC_EtDiagExtToString := 'HardwareException';
	ET_DiagExt.InvalidConfiguredParameter:		FC_EtDiagExtToString := 'InvalidConfiguredParameter';
	ET_DiagExt.TimeoutControlEnable:			FC_EtDiagExtToString := 'TimeoutControlEnable';
	ET_DiagExt.SegmentNotEnabled:				FC_EtDiagExtToString := 'SegmentNotEnabled';
	
ELSE
	FC_EtDiagExtToString := CONCAT('Unkown ET_DiagExt ', UDINT_TO_STRING(i_etDiagExt));
		
	q_etDiag	:= GD.ET_Diag.InputParameterInvalid;
	q_etDiagExt	:= ET_DiagExt.UnknownDiagExt;
END_CASE

END_FUNCTION

// LMC_PacDrive/Application/TemplateFullProgrammingFramework/EquipmentModules/SR_AlphaModule
PROGRAM SR_AlphaModule

VAR CONSTANT
(* Standard related constants *)
	c_udiNumberOfGroups				: UDINT := 0;			(* Maximum number of groups *)
	c_udiNumberOfGroupMembers		: UDINT := 0;			(* Maximum number of members per group *)

	c_udiNumberOfCmdTables			: UDINT := 8;			(* Must be the exact number of used CmdTables! *)
	c_udiNumberOfCmdSteps			: UDINT := 16;			(* Make sure that the number of command steps that each table
															   contains does not exceed the c_diNumberOfCmdSteps variable. *)

(* Definition group of modules *)
	c_udiAlphaGroup1				: UDINT := 2001;		(* Name of module group  1 *)
	c_udiAlphaGroup2				: UDINT := 2002;		(* Name of module group  2 *)

(* System generated code, could be modified for your application *)
	c_udiNumberOfSubModules			: UDINT := 1;			(* Number of SubModules *)
	c_udiMaster						: UDINT := 1;
(* End of system generated code, could be modified for your application *)
END_VAR

VAR (* User specific variables *)
	stMasterInterface				: AXM.ST_ModuleInterface;
	fbMasterModule					: AXM.FB_AxisModule;

	fbAxisModuleController			: AXM.FB_AxisModuleController;

END_VAR

VAR_INPUT
(* Master of AlphaModule *)
	i_ifMaster						: SystemConfigurationItf.IF_Master;
END_VAR

VAR_IN_OUT
(* TPL.ST_StandardModuleInterface *)	
	iq_stStandardModuleItf			: TPL.ST_StandardModuleInterface;
	
(* TPL.ST_StandardMotionInterface *)		
	iq_stStandardMotionItf			: TPL.ST_StandardMotionInterface;
	
(* ExceptionHandling and Logging *)	
	iq_stExceptionList				: TPL.ST_ExceptionList;
	iq_stLogDataList				: TPL.ST_LogDataList;
END_VAR

VAR
	xInitSuccessful : BOOL := TRUE;
	
(* Standard related variables *)
	astSubModuleInterface			: ARRAY[1..c_udiNumberOfSubModules] OF TPL.ST_StandardModuleInterface;		(* Interface to modules *)
	aaudiSubModuleGroups			: ARRAY[1..c_udiNumberOfGroups,1..c_udiNumberOfGroupMembers] OF UDINT;
	adwSubModuleAddInterfaces		: ARRAY[1..c_udiNumberOfSubModules] OF DWORD;

(* Modules related variables *)
	fbModuleController				: TPL.FB_ModuleController;
	etDiagModuleController			: GD.ET_Diag;
	etDiagExtModuleController		: TPL.ET_DiagExt;
	sMsgModuleController			: STRING[80];
	xWaitForStartStep				: BOOL;
	
	astListOfCmdTables				: ARRAY [1..c_udiNumberOfCmdTables] OF TPL.ST_CmdTable;
	udiTableIndex					: UDINT;
	udiStepIndex					: UDINT;
	diStep							: DINT;

	astPrepareTable					: ARRAY [1..c_udiNumberOfCmdSteps] OF TPL.ST_Cmd;		(* Relating Cmd table *)
	astAutoTable					: ARRAY [1..c_udiNumberOfCmdSteps] OF TPL.ST_Cmd;		(* Relating Cmd table *)
	astManualTable					: ARRAY [1..c_udiNumberOfCmdSteps] OF TPL.ST_Cmd;		(* Relating Cmd table *)
	astHoldTable					: ARRAY [1..c_udiNumberOfCmdSteps] OF TPL.ST_Cmd;		(* Relating Cmd table *)
	astStartTable					: ARRAY [1..c_udiNumberOfCmdSteps] OF TPL.ST_Cmd;		(* Relating Cmd table *)
	astStopTable					: ARRAY [1..c_udiNumberOfCmdSteps] OF TPL.ST_Cmd;		(* Relating Cmd table *)
	astBrakeReleaseTable			: ARRAY [1..c_udiNumberOfCmdSteps] OF TPL.ST_Cmd;		(* Relating Cmd table *)
	astAbortTable					: ARRAY [1..c_udiNumberOfCmdSteps] OF TPL.ST_Cmd;		(* Relating Cmd table *)

(* ExceptionHandling related variables *)
	fbExceptionHandler				: TPL.FB_ExceptionHandler2;

	aetReactionTranslationMode		: ARRAY[1..c_udiNumberOfSubModules] OF TPL.ET_ReactionTranslationMode;
	aastReactionTranslationTable	: ARRAY[1..c_udiNumberOfSubModules,1..TPL.Gc_udiMaxNumberOfReactions] OF TPL.ST_Reaction;
	astReactionTranslationJobs		: ARRAY[1..c_udiNumberOfSubModules] OF TPL.ST_ReactionTranslationJobs;

(* Exception declaration *)
	stUserException1				: TPL.ST_Exception;
	stUserException2				: TPL.ST_Exception;
	xModuleUserException1			: BOOL;
	xModuleUserException2			: BOOL;
	
	stUpdateStructsException		: TPL.ST_Exception;
	xUpdateStructsException			: BOOL;
	
	stInitReactionsException		: TPL.ST_Exception;
	xInitReactionsException			: BOOL;
	
	stInitSubModulesException		: TPL.ST_Exception;
	xInitSubModulesException		: BOOL;
	
	stIsDriveVirtualException		: TPL.ST_Exception;
	xIsDriveVirtualException		: BOOL;

(* Logging related variables*)
	fbLogger						: TPL.FB_Logger;
	fbLoggerPoint					: APL.FB_LoggerPoint;

(* OnlineChange related variables *)
	fbDetectOnlineChange			: TPL.FB_DetectOnlineChange;
	xDetectOnlineChangeActive		: BOOL; 
	xDetectOnlineChangeReady		: BOOL; 
	etDetectOnlineChangeDiag		: GD.ET_Diag;
	etDetectOnlineChangeDiagExt		: TPL.ET_DiagExt; 
	sDetectOnlineChangeMsg			: STRING[80];
	
(* Init related variables *)	
	stLogicalAddressMaster			: SystemConfigurationItf.ST_LogicalAddress;
	lrShaftRefDelay					: LREAL;
	iPositionDelay					: INT; 
	diResult						: DINT;

	xDriveIsVirtual					: BOOL;	
	
(* POU-Feedback related variables*)	
	etDiag			: GD.ET_Diag;
	etDiagExt		: ET_DiagExt;
	etDiagExtTPL	: TPL.ET_DiagExt;
	etDiagExtAXM	: AXM.ET_DiagExt;
	sMsgBuffer		: STRING[80];
	xReInit			: BOOL; 
	
(* Check RTB  *)
	diStateRTB						: DINT := 0;
	xRTBFailureFlag					: BOOL;
	udiCount						: UDINT;
	xModulesActive					: BOOL;
	xModulesNotActive				: BOOL;		
	
END_VAR

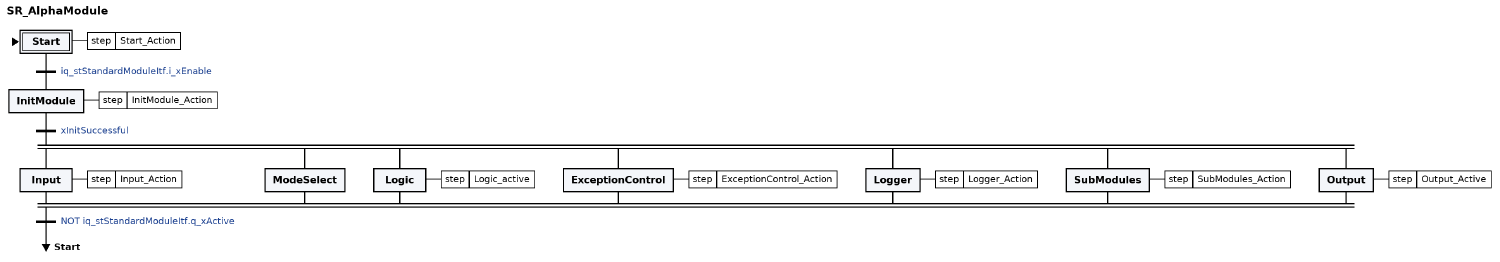
INITIAL_STEP Start:
    Start_Action(N);  // step action
END_STEP
TRANSITION FROM Start TO InitModule
    := iq_stStandardModuleItf.i_xEnable;
END_TRANSITION
STEP InitModule:
    InitModule_Action(N);  // step action
END_STEP
TRANSITION FROM InitModule TO (Input, ModeSelect, Logic, ExceptionControl, Logger, SubModules, Output)
    := xInitSuccessful;
END_TRANSITION
STEP Input:
    Input_Action(N);  // step action
END_STEP
STEP ModeSelect:
END_STEP
STEP Logic:
    Logic_active(N);  // step action
END_STEP
STEP ExceptionControl:
    ExceptionControl_Action(N);  // step action
END_STEP
STEP Logger:
    Logger_Action(N);  // step action
END_STEP
STEP SubModules:
    SubModules_Action(N);  // step action
END_STEP
STEP Output:
    Output_Active(N);  // step action
END_STEP
TRANSITION FROM (Input, ModeSelect, Logic, ExceptionControl, Logger, SubModules, Output) TO Start
    := NOT iq_stStandardModuleItf.q_xActive;
END_TRANSITION

ACTION Check_RTB:
(*
check RTB State
If RTB failure, all axis modules will be disabled.
After restart RTB, then all axis modules will be enabled again and the axes positions will be restored.
after home ok, opmode could be selected 
*)
(*########################################################################################*)

(* check RTB failure *)
IF Sercos_Master.State <> 4
AND NOT xRTBFailureFlag THEN

	xRTBFailureFlag := TRUE;
	
		(* disable axes modules *)
		FOR udiCount := 1 TO c_udiNumberOfSubModules DO
			
			(* axis module detection *)
			IF astSubModuleInterface[udiCount].q_dwModuleType = TPL.ET_ModuleType.AxisModule THEN
				astSubModuleInterface[udiCount].i_xEnable 		:= FALSE;	(* disable axes modules *)
			END_IF
		END_FOR
		
		diStateRTB := 10;

ELSIF Sercos_Master.State = 4 THEN	(* RTB ok *)
	xRTBFailureFlag := FALSE;
END_IF

(************************************************************************************************************************)
	CASE diStateRTB OF

	0:;	(* wait *)

	10:	(* wait for restart RTB *)

		IF Sercos_Master.State > 0
		AND Sercos_Master.State  <> 4 THEN
			xReInit								 := TRUE;		(* set marker reinit active *)
			diStateRTB := 20;
		END_IF

	20:	(* wait for RTB ready and ErrorQuit. / wait till AxesModules are disabled / --> restart axes modules *)
		FOR udiCount := 1 TO c_udiNumberOfSubModules DO
			
			(* axis module detection *)
			IF astSubModuleInterface[udiCount].q_dwModuleType = TPL.ET_ModuleType.AxisModule THEN
				IF astSubModuleInterface[udiCount].q_xActive THEN	(* module active *)
					xModulesNotActive 							:= FALSE;
					EXIT;
				ELSIF NOT astSubModuleInterface[udiCount].q_xActive THEN	(* module not active *)
					xModulesNotActive 							:= TRUE;
				END_IF
			END_IF
		END_FOR

		IF Sercos_Master.State = 4
		AND xModulesNotActive
		AND iq_stStandardModuleItf.i_xDiagQuit THEN
		
			FOR udiCount := 1 TO c_udiNumberOfSubModules DO
				(* axis module detection *)
				IF astSubModuleInterface[udiCount].q_dwModuleType = TPL.ET_ModuleType.AxisModule THEN
					astSubModuleInterface[udiCount].i_xEnable	 := TRUE;	(* enable axes modules *)
				END_IF
			END_FOR
			diStateRTB := 30;
		END_IF

	30:	(* wait for axes modules active *)

		FOR udiCount := 1 TO c_udiNumberOfSubModules DO
			
			(* axis module detection *)
			IF astSubModuleInterface[udiCount].q_dwModuleType = TPL.ET_ModuleType.AxisModule THEN
				IF NOT astSubModuleInterface[udiCount].q_xActive THEN	(* module not active *)
					xModulesActive 								:= FALSE;
					EXIT;
				ELSIF astSubModuleInterface[udiCount].q_xActive THEN	(* module active *)
					xModulesActive 								:= TRUE;
				END_IF
			END_IF
		END_FOR

		IF xModulesActive THEN	(* all axis modules active *)
			diStateRTB := 40;
		END_IF

	40:	(* Reinit ready  *)

		xReInit									:= FALSE;		(* reset marker reinit active *)
		diStateRTB := 0;

	END_CASE
END_ACTION

ACTION Init_Master:
//--- System generated code, could be modified for your application ---------------------------------------------------------

//--- Standard interface ---------------------------------------------------------
	//
	astSubModuleInterface[c_udiMaster].i_sModuleName	:= STANDARD.CONCAT(STR1 := iq_stStandardModuleItf.i_sModuleName, STR2 := ': Master');
	
	astSubModuleInterface[c_udiMaster].i_xLogEnable		:= TRUE;
	astSubModuleInterface[c_udiMaster].i_wLogDataFilter	:= UDINT_TO_WORD(TPL.ET_LogDataFilter.ModuleDefault);
	
	fbMasterModule.RegisterLoggerPoint(	i_ifParent	:= fbLoggerPoint,
										i_sName		:= 'Master',
										q_etDiag	:= ,
										q_etDiagExt	:= );

//
//--- Master, Drive& LEnc ---------------------------------------------------------
	//
	stMasterInterface.stMain.i_ifMaster		:= i_ifMaster; 		(* Master *)
	stMasterInterface.stMain.i_ifDrive		:= DRV_Master;
	stMasterInterface.stMain.iq_lencEncoder	:= LE_Master;	
//
//--- Check if Drive is virtual ---------------------------------------------------------
	//
	xDriveIsVirtual := FC_IsDriveVirtual(	i_ifDrive	:= stMasterInterface.stMain.i_ifDrive,
											q_etDiag	=> etDiag,
											q_etDiagExt	=> etDiagExt,
											q_sMsg		=> sMsgBuffer);
	
	IF etDiag <> GD.ET_Diag.Ok AND NOT xIsDriveVirtualException THEN										
		stIsDriveVirtualException.etDiag 	:= etDiag;
		stIsDriveVirtualException.udiDiagExt:= etDiagExt;
		stIsDriveVirtualException.sDiagExt 	:= FC_EtDiagExtToString(etDiagExt);										
		stIsDriveVirtualException.sMsg 		:= sMsgBuffer;
		xIsDriveVirtualException 			:= TRUE;
	END_IF
	
	fbExceptionHandler.SetException(i_xExceptionActive	:= xIsDriveVirtualException, 
									iq_stException		:= stIsDriveVirtualException, 
									iq_stExceptionList	:= iq_stExceptionList);
						
	xInitSuccessful := xInitSuccessful AND NOT xIsDriveVirtualException;
	etDiag := GD.ET_Diag.Ok;
	
//
//--- Set DeadTime compensation parameters depending on used type of Master ---------------------------------------------------------
	FC_SetDeadTimeCompensation(i_stSubModuleInterfaceMain := stMasterInterface.stMain);

//
//--- Set Velocity Parameters ---------------------------------------------------------
	stMasterInterface.stMain.i_lrMotionActiveVelLimit						:= 15.0;		(* Limit for max. velocity of astAxisModuleInterface to switch output AxisMove in Units/s *)
	stMasterInterface.stMain.i_etMotionActiveVelType						:= AXM.ET_MotionActiveVelType.Velocity;
	
	stMasterInterface.stMain.stReducedVelocity.i_xEnableReducedVelocity		:= FALSE;
	stMasterInterface.stMain.stReducedVelocity.i_xOnlyLimitCheck			:= FALSE;
	stMasterInterface.stMain.stReducedVelocity.i_lrMaxReducedVelocity		:= 50.0;
//
//--- Stop Parameters ---------------------------------------------------------
	stMasterInterface.stMain.i_timMasterStop								:= T#1S;
	stMasterInterface.stMain.i_xHwLimitPos									:= FALSE;
	stMasterInterface.stMain.i_xHwLimitNeg									:= FALSE;
	
	
	stMasterInterface.stMain.i_xStart										:= FALSE;

//
//--- Set Homing Mode ---------------------------------------------------------
	//
	IF xDriveIsVirtual THEN
		stMasterInterface.stHome.i_etMode := PDL.ET_HomeMode.SetPosAxisAndLogEncoderPosition;		(* Homing Mode in case of virtual axis *)
	ELSE
		stMasterInterface.stHome.i_etMode := PDL.ET_HomeMode.PosDirectionPosEdgeTp;					(* Homing Mode in case of real axis *)
	END_IF


	stMasterInterface.stHome.i_xEnableInitAbsReadPos := FALSE;						(* TRUE : Restores the AxisPosition depending on the stHome.etMode
																							  If stHome.i_etMode is equal to PDL.ET_HomeMode.RestorePosFromAxisEncoder or 
																							  to PDL.ET_HomeMode.WriteAxisEncoder, the encoder of the axis is read,
																							  or else the position will be restored from the retain area *)
	
	stMasterInterface.stHome.stSetpos.iq_pstRestorePosRetain := ADR(Grp_stRestorePositionAxis1);
	
	stMasterInterface.stHome.i_xResetHomeOk := FALSE;

//
//--- Homing mode Sensor:
	(*	PDL.ET_HomeMode.PosDirectionPosEdgeSensor
		PDL.ET_HomeMode.NegDirectionPosEdgeSensor
		PDL.ET_HomeMode.NegDirectionNegEdgeSensor
		PDL.ET_HomeMode.PosDirectionNegEdgeSensor	*)

	stMasterInterface.stHome.stSensor.i_lrHomePosition			:= 0.0;			(* Position at the end of homing in units *)
	stMasterInterface.stHome.stSensor.i_lrVel					:= 10.0;		(* Homing ceiling velocity in units/s *)
	stMasterInterface.stHome.stSensor.i_lrAcc					:= 1000.0;		(* Homing acceleration in units/s^2 *)
	stMasterInterface.stHome.stSensor.i_lrDec					:= 1000.0;		(* Homing deceleration in units/s^2 *)
	stMasterInterface.stHome.stSensor.i_lrJerk					:= 10000.0;		(* Homing jerk in units/s^3 *)
	stMasterInterface.stHome.stSensor.i_lrOffset				:= 0.0;			(* Offset from home signal in units *)
	stMasterInterface.stHome.stSensor.i_lrMaxTravel 			:= 720.0;		(* Max. travel for referencing by normal input *)
	stMasterInterface.stHome.stSensor.i_xRotativeSystem			:= FALSE;		(* Rotative system true or false for referencing by normal input *)
	stMasterInterface.stHome.stSensor.i_xSensor 				:= FALSE;		(* Input for home signal. Can be a signal from a controller input. Has to be written cyclic. *)

//--- Homing mode LimitSwitch:
	(* Possible Modes for homing mode LimitSwitch:
		PDL.ET_HomeMode.PosDirectionPosEdgeHWLimitPos		normally open contact / Closing contact
		PDL.ET_HomeMode.NegDirectionPosEdgeHWLimitNeg		normally open contact / Closing contact
		PDL.ET_HomeMode.NegDirectionNegEdgeHWLimitNeg		normally closed contact / Opening contact  
		PDL.ET_HomeMode.PosDirectionNegEdgeHWLimitPos		normally closed contact / Opening contact 
	*)
	stMasterInterface.stHome.stLimitSwitch.i_lrHomePosition 	:= 0.0;			(* Position at the end of homing in units *)
	stMasterInterface.stHome.stLimitSwitch.i_lrVel				:= 10.0;		(* Homing ceiling velocity in units/s *)
	stMasterInterface.stHome.stLimitSwitch.i_lrLowVel			:= 5.0;			(* Homing low ceiling velocity in units/s *)
	stMasterInterface.stHome.stLimitSwitch.i_lrAcc				:= 1000.0;		(* Homing acceleration in units/s^2 *)
	stMasterInterface.stHome.stLimitSwitch.i_lrDec				:= 1000.0;		(* Homing deceleration in units/s^2 *)
	stMasterInterface.stHome.stLimitSwitch.i_lrJerk				:= 10000.0;		(* Homing jerk in units/s^3 *)
	stMasterInterface.stHome.stLimitSwitch.i_lrOffset			:= 0.0;			(* Offset from home signal in units *)
	stMasterInterface.stHome.stLimitSwitch.i_lrMaxTravel 		:= 9999.0;		(* Max. travel for referencing normal input as a hardware limit *)

//--- Homing mode MoveOnPos:
	(* Possible modes for homing mode MoveOnPos:
		PDL.ET_HomeMode.MoveOnPosAbs 
	*)
	stMasterInterface.stHome.stMoveOnPos.i_lrTarget				:= 0.0;			(* Position at the end of homing in units *)
	stMasterInterface.stHome.stMoveOnPos.i_lrVel				:= 10.0;		(* Homing ceiling velocity in units/s *)
	stMasterInterface.stHome.stMoveOnPos.i_lrAcc				:= 1000.0;		(* Homing acceleration in units/s^2 *)
	stMasterInterface.stHome.stMoveOnPos.i_lrDec				:= 1000.0;		(* Homing deceleration in units/s^2 *)
	stMasterInterface.stHome.stMoveOnPos.i_lrJerk				:= 10000.0;		(* Homing jerk in units/s^3 *)
	stMasterInterface.stHome.stMoveOnPos.i_lrPeriod				:= 0.0;			(* Period of the axis *)
	stMasterInterface.stHome.stMoveOnPos.i_xRotativeSystem		:= FALSE;		(* Rotative system true or false *)

//--- Homing mode SetPos:
	(* Possible modes for homing mode SetPos:
		PDL.ET_HomeMode.SetPosAxisPosition 
		PDL.ET_HomeMode.SetPosLogEncoderPosition 
		PDL.ET_HomeMode.SetPosAxisAndLogEncoderPosition
		PDL.ET_HomeMode.RestorePosFromAxisEncoder 
		PDL.ET_HomeMode.RestorePosFromRetain 
	*)
	stMasterInterface.stHome.stSetpos.i_lrHomePosition			:= 0.0;			(* Position at the end of homing in units *)
	stMasterInterface.stHome.stSetpos.i_lrEncoderPosition		:= 0.0;			(* Encoder position in units after homing *)
	stMasterInterface.stHome.stSetpos.i_lrAbsEncOffset			:= 100.0;		(* Distance to the jump of axis encoder in units *)
	stMasterInterface.stHome.stSetpos.i_lrRestoreWindow			:= 180;			(* How far can the drive be away from its correct position *)
	stMasterInterface.stHome.stSetpos.i_lrUserPeriod			:= 360;			(* Period of the axis *)

//--- Homing mode Torque:
	(* Possible modes for homing mode Torque:
		PDL.ET_HomeMode.PosDirectionMaxTorque 
		PDL.ET_HomeMode.NegDirectionMaxTorque 
	*)
	stMasterInterface.stHome.stTorque.i_lrHomePosition			:= 0.0;			(* Position at the end of homing in units *)
	stMasterInterface.stHome.stTorque.i_lrVel					:= 10.0;		(* Homing ceiling velocity in units/s *)
	stMasterInterface.stHome.stTorque.i_lrAcc					:= 1000.0;		(* Homing acceleration in units/s^2 *)
	stMasterInterface.stHome.stTorque.i_lrDec					:= 1000.0;		(* Homing deceleration in units/s^2 *)
	stMasterInterface.stHome.stTorque.i_lrJerk					:= 10000.0;		(* Homing jerk in units/s^3 *)
	stMasterInterface.stHome.stTorque.i_lrOffset				:= 0.0;			(* Offset from home signal in units *)
	stMasterInterface.stHome.stTorque.i_lrMaxTravel				:= 9999.0;		(* Max. travel for referencing by torque *)
	stMasterInterface.stHome.stTorque.i_lrMaxTorque				:= 0.0;			(* Torque for stop in Nm / referencing by torque *)
	stMasterInterface.stHome.stTorque.i_diTorqueTime			:= 5;			(* Time in msec to hold torque *)

//--- Homing mode TouchProbe:
	(* Possible modes for homing mode TouchProbe:
		PDL.ET_HomeMode.PosDirectionPosEdgeTp 
		PDL.ET_HomeMode.NegDirectionPosEdgeTp 
		PDL.ET_HomeMode.NegDirectionNegEdgeTp 
		PDL.ET_HomeMode.PosDirectionNegEdgeTp 
	*)
	stMasterInterface.stHome.stTouchProbe.i_lrHomePosition		:= 0.0;			(* Position at the end of homing in units *)
	stMasterInterface.stHome.stTouchProbe.i_lrVel				:= 100.0;		(* Homing ceiling velocity in units/s *)
	stMasterInterface.stHome.stTouchProbe.i_lrAcc				:= 1000.0;		(* Homing acceleration in units/s^2 *)
	stMasterInterface.stHome.stTouchProbe.i_lrDec				:= 1000.0;		(* Homing deceleration in units/s^2 *)
	stMasterInterface.stHome.stTouchProbe.i_lrJerk				:= 10000.0;		(* Homing jerk in units/s^3 *)
	stMasterInterface.stHome.stTouchProbe.i_lrOffset			:= 30.0;		(* Offset from home signal in units *)
	stMasterInterface.stHome.stTouchProbe.i_lrMaxTravel			:= 720.0;		(* Max. travel for referencing by TP *)
	stMasterInterface.stHome.stTouchProbe.i_xRotativeSystem		:= TRUE;		(* Rotative system true or false for referencing by TP *)
	stMasterInterface.stHome.stTouchProbe.i_ifTouchProbe		:= TP_0;		(* Input for TP *)

//--- Homing mode WritePos:
	(* Possible modes for homing mode WritePos:
		PDL.ET_HomeMode.WriteAxisEncoder 
	*)
	stMasterInterface.stHome.stWritePos.i_lrHomePosition		:= 0.0;			(* Position at the end of homing in units *)
	stMasterInterface.stHome.stWritePos.i_lrUserPeriod			:= 0.0;			(* Calculates Drive.Position into period ( units ) *)
	stMasterInterface.stHome.stWritePos.i_lrAbsEncOffset		:= 100.0;		(* Distance to the jump of axis encoder in units *)

//
//--- Manual ---------------------------------------------------------
	//
	stMasterInterface.stManual.i_lrVel								:= 50.0;			(* Velocity in units/s *)
	stMasterInterface.stManual.i_lrAcc								:= 100.0;			(* Acceleration in units/s^2 *)
	stMasterInterface.stManual.i_lrDec								:= 100.0;			(* Deceleration in units/s^2 *)
	stMasterInterface.stManual.i_lrJerk								:= 1000.0;			(* Jerk in units/s^3 *)
	stMasterInterface.stManual.i_lrMaxDistance						:= 120.0;			(* Max pathlengths for one step in units *)
	stMasterInterface.stManual.i_xEndless							:= FALSE;			(* TRUE: jogging endless; Position between the periode; FALSE: jogging in steps. Position can be out of periode *)
	stMasterInterface.stManual.i_lrPeriod							:= 360.0;			(* Period of the axis *)

//
//--- Cam ---------------------------------------------------------
	//
	stMasterInterface.stMultiCam.i_etCSModeSlave					:= PDL.ET_MultiCamCsModeSlave.SetSlavePositionToFirstCamPosition;		(* ColdStartMode Slave *)
	stMasterInterface.stMultiCam.i_etCSModeMaster					:= PDL.ET_MultiCamCsModeMaster.SetMasterPositionToFirstCamPosition;		(* ColdStartMode Master *)
	stMasterInterface.stMultiCam.i_etWSMode							:= PDL.ET_MultiCamWsMode.StoredCamMoveAlwaysNoPositionCheck;			(* WarmStartMode *)
	stMasterInterface.stMultiCam.i_lrWSWindow						:= 5.0;											(* WarmStartWindow in Axis units *)
	stMasterInterface.stMultiCam.i_lrWSVel							:= 10.0;										(* Velocity for WarmStart and CSModeSlave = PDL.ET_MultiCamCsModeSlave.MoveSlaveToFirstCamPosition in Units/s *)
	stMasterInterface.stMultiCam.i_lrWSAcc							:= 1000.0;										(* Acceleration and deceleration for Warmstart and CSModeSlave = PDL.ET_MultiCamCsModeSlave.MoveSlaveToFirstCamPosition in Units/s^2 *)
	stMasterInterface.stMultiCam.i_lrWSJerk							:= 10000.0;										(* Jerk for Warmstart and CSModeSlave = PDL.ET_MultiCamCsModeSlave.MoveSlaveToFirstCamPosition in units/s^3 *)
	stMasterInterface.stMultiCam.i_diTXend							:= 2*SYSTEMINTERFACE.FC_LzsTaskGetInterval();	(* Time of XLowEnd and XHighEnd befor Xend or Xstart in msec*)
	stMasterInterface.stMultiCam.i_lrInstantXLimMax					:= 0.0;											(* Switch off position at 'InstantNewCam' *)
	
	stMasterInterface.stMultiCam.i_xEnableTabHandler				:= TRUE;										(* TRUE: TabHandler is enabled *)
	stMasterInterface.stMultiCam.i_udiTableSelectNr					:= AXM.ET_ParId.User;							(* Number of table which is used in the next cycle *)								
	
	stMasterInterface.stMultiCam.i_xSetEncoderParameters			:= FALSE;										(* TRUE: The parameters MasterId, FeedConstand, GearIn and GearOut will be copyed into LEnc object *)
	stMasterInterface.stMultiCam.i_xSetEncoderPosition				:= TRUE;										(* TRUE: Manipulation of LEnc object on startup OpMode MultiCam *)
	stMasterInterface.stMultiCam.i_lrSetEncoderOffset				:= 0.0;											(* Master encoder offset *)
	stMasterInterface.stMultiCam.i_xCheckEncoderPeriod				:= TRUE;										(* TRUE: Check of encoder period = 0. If encoder period <> 0 -> Exception *)
	
	// stMasterInterface.stMultiCam.iq_xNewCam						:= FALSE;										(* TRUE: A new DataStruct will be load for next cycle. Will be reset when new cycle is started in case of stMultiCam.i_xEnableTabHandler = FALSE. *)
	// stMasterInterface.stMultiCam.iq_xInstantNewCam				:= FALSE;										(* TRUE: A new DataStruct will be load. It will be active at master position stMultiCam.i_lrInstantXLimMax. Will be reset when ne DataStruct is active *)
	// stMasterInterface.stMultiCam.iq_xChangeMaster				:= FALSE;										(* TRUE: Switch to a new Master. Will be reset when done. *)			
	
	// stMasterInterface.stMultiCam.iq_stExt		;						(* Extended In of the Multicam FB, can be used if needed! *)
	
	stMasterInterface.stMultiCam.iq_astMotionPar[AXM.ET_ParId.User].diNumberOfCamPoints			:= 4;	(* DataStruct for the next cycle *)
	stMasterInterface.stMultiCam.iq_astMotionPar[AXM.ET_ParId.User].lrYPeriod					:= 0.0;
	
	stMasterInterface.stMultiCam.iq_astMotionPar[AXM.ET_ParId.User].astCamPoint[0].lrX			:= 0.0;
	stMasterInterface.stMultiCam.iq_astMotionPar[AXM.ET_ParId.User].astCamPoint[0].lrY			:= 0.0;
	stMasterInterface.stMultiCam.iq_astMotionPar[AXM.ET_ParId.User].astCamPoint[0].lrM			:= 0.0;
	stMasterInterface.stMultiCam.iq_astMotionPar[AXM.ET_ParId.User].astCamPoint[0].etCamType	:= PDL.ET_CamType.Poly5Com;
	stMasterInterface.stMultiCam.iq_astMotionPar[AXM.ET_ParId.User].astCamPoint[1].lrX			:= 60.0;
	stMasterInterface.stMultiCam.iq_astMotionPar[AXM.ET_ParId.User].astCamPoint[1].lrY			:= 30.0;
	stMasterInterface.stMultiCam.iq_astMotionPar[AXM.ET_ParId.User].astCamPoint[1].lrM			:= 1.0;
	stMasterInterface.stMultiCam.iq_astMotionPar[AXM.ET_ParId.User].astCamPoint[1].etCamType	:= PDL.ET_CamType.Straight;
	stMasterInterface.stMultiCam.iq_astMotionPar[AXM.ET_ParId.User].astCamPoint[2].lrX			:= 240.0;
	stMasterInterface.stMultiCam.iq_astMotionPar[AXM.ET_ParId.User].astCamPoint[2].lrY			:= 210.0;
	stMasterInterface.stMultiCam.iq_astMotionPar[AXM.ET_ParId.User].astCamPoint[2].lrM			:= 1.0;
	stMasterInterface.stMultiCam.iq_astMotionPar[AXM.ET_ParId.User].astCamPoint[2].etCamType	:= PDL.ET_CamType.Poly5Com;
	stMasterInterface.stMultiCam.iq_astMotionPar[AXM.ET_ParId.User].astCamPoint[3].lrX			:= 360.0;
	stMasterInterface.stMultiCam.iq_astMotionPar[AXM.ET_ParId.User].astCamPoint[3].lrY			:= 0.0;
	stMasterInterface.stMultiCam.iq_astMotionPar[AXM.ET_ParId.User].astCamPoint[3].lrM			:= 0.0;
	stMasterInterface.stMultiCam.iq_astMotionPar[AXM.ET_ParId.User].astCamPoint[3].etCamType	:= PDL.ET_CamType.Poly5Com;
	
	stMasterInterface.stMultiCam.iq_astMotionPar[AXM.ET_ParId.Idle].diUserTableId	:= UDINT_TO_DINT(AXM.ET_ParId.Idle);
	stMasterInterface.stMultiCam.iq_astMotionPar[AXM.ET_ParId.Start].diUserTableId	:= UDINT_TO_DINT(AXM.ET_ParId.Start);
	stMasterInterface.stMultiCam.iq_astMotionPar[AXM.ET_ParId.Cont].diUserTableId	:= UDINT_TO_DINT(AXM.ET_ParId.Cont);
	stMasterInterface.stMultiCam.iq_astMotionPar[AXM.ET_ParId.Stop].diUserTableId	:= UDINT_TO_DINT(AXM.ET_ParId.Stop);
	stMasterInterface.stMultiCam.iq_astMotionPar[AXM.ET_ParId.User].diUserTableId	:= UDINT_TO_DINT(AXM.ET_ParId.User);
	
	
	//--- ILS Data --------------------------------------------------------
	//---
	// 	stMasterInterface.stMultiCam.i_udiIlsSlaveNumber														:= 1;
	// 	
	// 	G_stIlsData.i_stRunTime.astSlaveLimits[stMasterInterface.stMultiCam.i_udiIlsSlaveNumber].lrPosVel	:= 1000.0;
	// 	G_stIlsData.i_stRunTime.astSlaveLimits[stMasterInterface.stMultiCam.i_udiIlsSlaveNumber].lrNegVel	:= -1000.0;
	// 	G_stIlsData.i_stRunTime.astSlaveLimits[stMasterInterface.stMultiCam.i_udiIlsSlaveNumber].lrPosAcc	:= 10000.0;
	// 	G_stIlsData.i_stRunTime.astSlaveLimits[stMasterInterface.stMultiCam.i_udiIlsSlaveNumber].lrNegAcc	:= -10000.0;
	// 	
	// 	G_stIlsData.i_astCamData[stMasterInterface.stMultiCam.i_diIlsSlaveNumber].diNumberOfMasterPeriods	:= 1;	
	// 	G_stIlsData.i_astCamData[stMasterInterface.stMultiCam.i_diIlsSlaveNumber].diMasterPeriodInit		:= 1;
	// 	G_stIlsData.i_astCamData[stMasterInterface.stMultiCam.i_diIlsSlaveNumber].lrXOffset					:= 0.0;
	// 	
	// 	stMasterInterface.stMultiCam.pstIlsData																:= ADR(G_stIlsData);

//
//--- Endless ---------------------------------------------------------
	//
	stMasterInterface.stEndless.i_lrVel								:= 0.0;					(* Velocity in Units/s *)
	stMasterInterface.stEndless.i_lrAcc								:= 10_000.0;			(* Acceleration in Units/s^2 *)
	stMasterInterface.stEndless.i_lrDec								:= 10_000.0;			(* Deceleration in Units/s^2 *)
	stMasterInterface.stEndless.i_lrJerk							:= 100_000.0;			(* Jerk in units/s^3 *)
	stMasterInterface.stEndless.i_lrPeriod							:= 360.0;				(* Period one cycle in units *)
	stMasterInterface.stEndless.i_lrStopPosition					:= 0.5;					(* Stop position in units *)
	
//--- Endless ILS ---------------------------------------------------------
	//
	//G_stIlsData.i_stConfig.diNumberOfSlaves							:= 0;
	//G_stIlsData.i_stConfig.diPositionGridSize						:= 500;
	//G_stIlsData.i_stConfig.diTimeGridSize							:= 50;
	//G_stIlsData.i_stConfig.lrHysteresis								:= 20;
	//
	//G_stIlsData.i_stRunTime.iMasterAverageVelocityCycles			:= 10;
	//G_stIlsData.i_stRunTime.lrMasterMaxAbsVel						:= 100.0;
	//G_stIlsData.i_stRunTime.lrMasterMaxAbsAcc						:= 1000.0;
	//G_stIlsData.i_stRunTime.lrMasterMaxAbsJerk						:= 10000.0;
	//G_stIlsData.i_stRunTime.xActivateLimitation						:= TRUE;
	//
	//stSlave1Interface.stEndless.pstIlsData							:= ADR(G_stIlsData);
//
//--- Pos ---------------------------------------------------------
	//

	stMasterInterface.stPos.i_etPosMode								:= SYSTEMINTERFACE.ET_PosMode.Endless;		(* SYSTEMINTERFACE.ET_PosMode.Endless, SYSTEMINTERFACE.ET_PosMode.Relative, SYSTEMINTERFACE.ET_PosMode.Absolute *)
	stMasterInterface.stPos.i_lrTarget								:= 360.0;									(* Target position or distance in Units *)
	stMasterInterface.stPos.i_lrVel									:= 360.0;									(* Ceiling velocity in Units/s *)
	stMasterInterface.stPos.i_lrAcc									:= 3600.0;									(* Acceleration in Units/s^2 *)
	stMasterInterface.stPos.i_lrDec									:= 3600.0;									(* Deceleration in Units/s^2 *)
	stMasterInterface.stPos.i_lrJerk								:= 36000.0;									(* Jerk in units/s^3 *)
	
	//--- stMasterInterface.stPos.i_xStop								:= FALSE;
//
//--- End of system generated code, could be modified for your application ---------------------------------------------------------
END_ACTION

ACTION Init_CmdTables:
(* System generated code, could be modified for your application *)

//-------------------------------------------------------------------------------------------------------------------
//-- Prepare  --
	//
	TPL.FC_FirstStep(udiStepIndex, diStep);
	astPrepareTable[udiStepIndex].sTitle					:= 'DriveEnable On AllSubModules';
	astPrepareTable[udiStepIndex].udiModuleName				:= TPL.Gc_udiAllSubModules;
	astPrepareTable[udiStepIndex].diStep					:= diStep;
	astPrepareTable[udiStepIndex].diCMD						:= AXM.ET_Cmd.DriveEnableOn;
	astPrepareTable[udiStepIndex].timTimeOut				:= T#0MS;
	astPrepareTable[udiStepIndex].xEndCMD					:= FALSE;
	
	TPL.FC_NextStep(udiStepIndex, diStep);
	astPrepareTable[udiStepIndex].sTitle					:= 'Homing Mode AllSubModules';
	astPrepareTable[udiStepIndex].udiModuleName				:= TPL.Gc_udiAllSubModules;
	astPrepareTable[udiStepIndex].diStep					:= diStep;
	astPrepareTable[udiStepIndex].diCMD						:= AXM.ET_Cmd.Homing;
	astPrepareTable[udiStepIndex].timTimeOut				:= T#0MS;
	astPrepareTable[udiStepIndex].xEndCMD					:= FALSE;
	
	TPL.FC_NextStep(udiStepIndex, diStep);
	astPrepareTable[udiStepIndex].sTitle					:= 'Start AllSubModules';
	astPrepareTable[udiStepIndex].udiModuleName				:= TPL.Gc_udiAllSubModules;
	astPrepareTable[udiStepIndex].diStep					:= diStep;
	astPrepareTable[udiStepIndex].diCMD						:= AXM.ET_Cmd.Start;
	astPrepareTable[udiStepIndex].timTimeOut				:= T#0MS;
	astPrepareTable[udiStepIndex].xEndCMD					:= FALSE;
	
	TPL.FC_LastStep(udiStepIndex, diStep);
	astPrepareTable[udiStepIndex].sTitle					:= 'End';
	astPrepareTable[udiStepIndex].udiModuleName				:= 0;
	astPrepareTable[udiStepIndex].diStep					:= diStep;
	astPrepareTable[udiStepIndex].diCMD						:= 0;
	astPrepareTable[udiStepIndex].timTimeOut				:= T#0MS;
	astPrepareTable[udiStepIndex].xEndCMD					:= TRUE;
	
	TPL.FC_FirstCmdTable(iq_udiTableIndex := udiTableIndex);
	astListofCMDTables[udiTableIndex].sTitle				:= 'Prepare';
	astListofCMDTables[udiTableIndex].diCMD					:= ET_Cmd.Prepare;
	astListofCMDTables[udiTableIndex].udiNumberOfCmdSteps	:= udiStepIndex;

//-------------------------------------------------------------------------------------------------------------------
//-- Auto  --
	//
	TPL.FC_FirstStep(udiStepIndex, diStep);
	astAutoTable[udiStepIndex].sTitle						:= 'DriveEnable On AllSubModules';
	astAutoTable[udiStepIndex].udiModuleName				:= TPL.Gc_udiAllSubModules;
	astAutoTable[udiStepIndex].diStep						:= diStep;
	astAutoTable[udiStepIndex].diCMD						:= AXM.ET_Cmd.DriveEnableOn;
	astAutoTable[udiStepIndex].timTimeOut					:= T#0MS;
	astAutoTable[udiStepIndex].xEndCMD						:= FALSE;
	
	TPL.FC_NextStep(udiStepIndex, diStep);
	astAutoTable[udiStepIndex].sTitle						:= 'Endless Mode AllSubModules';
	astAutoTable[udiStepIndex].udiModuleName				:= TPL.Gc_udiAllSubModules;
	astAutoTable[udiStepIndex].diStep						:= diStep;
	astAutoTable[udiStepIndex].diCMD						:= AXM.ET_Cmd.Endless;
	astAutoTable[udiStepIndex].timTimeOut					:= T#0MS;
	astAutoTable[udiStepIndex].xEndCMD						:= FALSE;
	
	TPL.FC_NextStep(udiStepIndex, diStep);
	astAutoTable[udiStepIndex].sTitle						:= 'Start AllSubModules';
	astAutoTable[udiStepIndex].udiModuleName				:= TPL.Gc_udiAllSubModules;
	astAutoTable[udiStepIndex].diStep						:= diStep;
	astAutoTable[udiStepIndex].diCMD						:= AXM.ET_Cmd.Start;
	astAutoTable[udiStepIndex].timTimeOut					:= T#0MS;
	astAutoTable[udiStepIndex].xEndCMD						:= FALSE;
	
	TPL.FC_LastStep(udiStepIndex, diStep);
	astAutoTable[udiStepIndex].sTitle						:= 'End';
	astAutoTable[udiStepIndex].udiModuleName				:= 0;
	astAutoTable[udiStepIndex].diStep						:= diStep;
	astAutoTable[udiStepIndex].diCMD						:= 0;
	astAutoTable[udiStepIndex].timTimeOut					:= T#0MS;
	astAutoTable[udiStepIndex].xEndCMD						:= TRUE;
	
	TPL.FC_NextCmdTable(iq_udiTableIndex:= udiTableIndex);
	astListofCMDTables[udiTableIndex].sTitle				:= 'Auto';
	astListofCMDTables[udiTableIndex].diCMD					:= ET_Cmd.Auto;
	astListofCMDTables[udiTableIndex].udiNumberOfCmdSteps	:= udiStepIndex;

//-------------------------------------------------------------------------------------------------------------------
//-- Manual  --
	//
	TPL.FC_FirstStep(udiStepIndex, diStep);
	astManualTable[udiStepIndex].sTitle						:= 'DriveEnable On AllSubModules';
	astManualTable[udiStepIndex].udiModuleName				:= TPL.Gc_udiAllSubModules;
	astManualTable[udiStepIndex].diStep						:= diStep;
	astManualTable[udiStepIndex].diCMD						:= AXM.ET_Cmd.DriveEnableOn;
	astManualTable[udiStepIndex].timTimeOut					:= T#0MS;
	astManualTable[udiStepIndex].xEndCMD					:= FALSE;
	
	TPL.FC_NextStep(udiStepIndex, diStep);
	astManualTable[udiStepIndex].sTitle						:= 'Manual Mode AllSubModules';
	astManualTable[udiStepIndex].udiModuleName				:= TPL.Gc_udiAllSubModules;
	astManualTable[udiStepIndex].diStep						:= diStep;
	astManualTable[udiStepIndex].diCMD						:= AXM.ET_Cmd.Manual;
	astManualTable[udiStepIndex].timTimeOut					:= T#0MS;
	astManualTable[udiStepIndex].xEndCMD					:= FALSE;
	
	TPL.FC_LastStep(udiStepIndex, diStep);
	astManualTable[udiStepIndex].sTitle						:= 'End';
	astManualTable[udiStepIndex].udiModuleName				:= 0;
	astManualTable[udiStepIndex].diStep						:= diStep;
	astManualTable[udiStepIndex].diCMD						:= 0;
	astManualTable[udiStepIndex].timTimeOut					:= T#0MS;
	astManualTable[udiStepIndex].xEndCMD					:= TRUE;
	
	TPL.FC_NextCmdTable(iq_udiTableIndex:= udiTableIndex);
	astListofCMDTables[udiTableIndex].sTitle				:= 'Manual';
	astListofCMDTables[udiTableIndex].diCMD					:= ET_Cmd.Manual;
	astListofCMDTables[udiTableIndex].udiNumberOfCmdSteps	:= udiStepIndex;

//-------------------------------------------------------------------------------------------------------------------
//-- Stop --
	//
	TPL.FC_FirstStep(udiStepIndex, diStep);
	astStopTable[udiStepIndex].sTitle						:= 'Stop AllSubModules';
	astStopTable[udiStepIndex].udiModuleName				:= TPL.Gc_udiAllSubModules;
	astStopTable[udiStepIndex].diStep						:= diStep;
	astStopTable[udiStepIndex].diCMD						:= AXM.ET_Cmd.Stop;
	astStopTable[udiStepIndex].timTimeOut					:= T#0MS;
	astStopTable[udiStepIndex].xEndCMD						:= FALSE;
	
	TPL.FC_LastStep(udiStepIndex, diStep);
	astStopTable[udiStepIndex].sTitle						:= 'End';
	astStopTable[udiStepIndex].udiModuleName				:= 0;
	astStopTable[udiStepIndex].diStep						:= diStep;
	astStopTable[udiStepIndex].diCMD						:= 0;
	astStopTable[udiStepIndex].timTimeOut					:= T#0MS;
	astStopTable[udiStepIndex].xEndCMD						:= TRUE;
	
	TPL.FC_NextCmdTable(iq_udiTableIndex:= udiTableIndex);
	astListofCMDTables[udiTableIndex].sTitle				:= 'Stop';
	astListofCMDTables[udiTableIndex].diCMD					:= ET_Cmd.Stop;
	astListofCMDTables[udiTableIndex].udiNumberOfCmdSteps	:= udiStepIndex;
	
//-------------------------------------------------------------------------------------------------------------------
//-- Start --
	//
	TPL.FC_FirstStep(udiStepIndex, diStep);
	astStartTable[udiStepIndex].sTitle						:= 'Start AllSubModules';
	astStartTable[udiStepIndex].udiModuleName				:= TPL.Gc_udiAllSubModules;
	astStartTable[udiStepIndex].diStep						:= diStep;
	astStartTable[udiStepIndex].diCMD						:= AXM.ET_Cmd.Start;
	astStartTable[udiStepIndex].timTimeOut					:= T#0MS;
	astStartTable[udiStepIndex].xEndCMD						:= FALSE;
	
	TPL.FC_LastStep(udiStepIndex, diStep);
	astStartTable[udiStepIndex].sTitle						:= 'End';
	astStartTable[udiStepIndex].udiModuleName				:= 0;
	astStartTable[udiStepIndex].diStep						:= diStep;
	astStartTable[udiStepIndex].diCMD						:= 0;
	astStartTable[udiStepIndex].timTimeOut					:= T#0MS;
	astStartTable[udiStepIndex].xEndCMD						:= TRUE;
	
	TPL.FC_NextCmdTable(iq_udiTableIndex:= udiTableIndex);
	astListofCMDTables[udiTableIndex].sTitle				:= 'Start';
	astListofCMDTables[udiTableIndex].diCMD					:= ET_Cmd.Start;
	astListofCMDTables[udiTableIndex].udiNumberOfCmdSteps	:= udiStepIndex;

//-------------------------------------------------------------------------------------------------------------------
//-- Abort --
	//
	TPL.FC_FirstStep(udiStepIndex, diStep);
	astAbortTable[udiStepIndex].sTitle						:= 'Stop AllSubModules';
	astAbortTable[udiStepIndex].udiModuleName				:= TPL.Gc_udiAllSubModules;
	astAbortTable[udiStepIndex].diStep						:= diStep;
	astAbortTable[udiStepIndex].diCMD						:= AXM.ET_Cmd.Stop;
	astAbortTable[udiStepIndex].timTimeOut					:= T#0MS;
	astAbortTable[udiStepIndex].xEndCMD						:= FALSE;
	
	TPL.FC_LastStep(udiStepIndex, diStep);
	astAbortTable[udiStepIndex].sTitle						:= 'End';
	astAbortTable[udiStepIndex].udiModuleName				:= 0;
	astAbortTable[udiStepIndex].diStep						:= diStep;
	astAbortTable[udiStepIndex].diCMD						:= 0;
	astAbortTable[udiStepIndex].timTimeOut					:= T#0MS;
	astAbortTable[udiStepIndex].xEndCMD						:= TRUE;
	
	TPL.FC_NextCmdTable(iq_udiTableIndex:= udiTableIndex);
	astListofCMDTables[udiTableIndex].sTitle				:= 'Abort';
	astListofCMDTables[udiTableIndex].diCMD					:= ET_Cmd.Abort;
	astListofCMDTables[udiTableIndex].udiNumberOfCmdSteps	:= udiStepIndex;

//-------------------------------------------------------------------------------------------------------------------
//-- Hold --
	//
	TPL.FC_FirstStep(udiStepIndex, diStep);
	astHoldTable[udiStepIndex].sTitle						:= 'Hold AllSubModules';
	astHoldTable[udiStepIndex].udiModuleName				:= TPL.Gc_udiAllSubModules;
	astHoldTable[udiStepIndex].diStep						:= diStep;
	astHoldTable[udiStepIndex].diCMD						:= AXM.ET_Cmd.Hold;
	astHoldTable[udiStepIndex].timTimeOut					:= T#0MS;
	astHoldTable[udiStepIndex].xEndCMD						:= FALSE;
	
	TPL.FC_LastStep(udiStepIndex, diStep);
	astHoldTable[udiStepIndex].sTitle						:= 'End';
	astHoldTable[udiStepIndex].udiModuleName				:= 0;
	astHoldTable[udiStepIndex].diStep						:= diStep;
	astHoldTable[udiStepIndex].diCMD						:= 0;
	astHoldTable[udiStepIndex].timTimeOut					:= T#0MS;
	astHoldTable[udiStepIndex].xEndCMD						:= TRUE;
	
	TPL.FC_NextCmdTable(iq_udiTableIndex:= udiTableIndex);
	astListofCMDTables[udiTableIndex].sTitle				:= 'Hold';
	astListofCMDTables[udiTableIndex].diCMD					:= ET_Cmd.Hold;
	astListofCMDTables[udiTableIndex].udiNumberOfCmdSteps	:= udiStepIndex;
//-------------------------------------------------------------------------------------------------------------------
//-- Brake Release --
	//
	TPL.FC_FirstStep(udiStepIndex, diStep);
	astBrakeReleaseTable[udiStepIndex].sTitle				:= 'DriveEnable Off AllSubModules';
	astBrakeReleaseTable[udiStepIndex].udiModuleName		:= TPL.Gc_udiAllSubModules;
	astBrakeReleaseTable[udiStepIndex].diStep				:= diStep;
	astBrakeReleaseTable[udiStepIndex].diCMD				:= AXM.ET_Cmd.DriveEnableOff;
	astBrakeReleaseTable[udiStepIndex].timTimeOut			:= T#0MS;
	astBrakeReleaseTable[udiStepIndex].xEndCMD				:= FALSE;
	
	TPL.FC_NextStep(udiStepIndex, diStep);
	astBrakeReleaseTable[udiStepIndex].sTitle				:= 'BrakeRelease Mode AllSubModules';
	astBrakeReleaseTable[udiStepIndex].udiModuleName		:= TPL.Gc_udiAllSubModules;
	astBrakeReleaseTable[udiStepIndex].diStep				:= diStep;
	astBrakeReleaseTable[udiStepIndex].diCMD				:= AXM.ET_Cmd.BrakeRelease;
	astBrakeReleaseTable[udiStepIndex].timTimeOut			:= T#0MS;
	astBrakeReleaseTable[udiStepIndex].xEndCMD				:= FALSE;
	
	TPL.FC_NextStep(udiStepIndex, diStep);
	astBrakeReleaseTable[udiStepIndex].sTitle				:= 'Start AllSubModules';
	astBrakeReleaseTable[udiStepIndex].udiModuleName		:= TPL.Gc_udiAllSubModules;
	astBrakeReleaseTable[udiStepIndex].diStep				:= diStep;
	astBrakeReleaseTable[udiStepIndex].diCMD				:= AXM.ET_Cmd.Start;
	astBrakeReleaseTable[udiStepIndex].timTimeOut			:= T#0MS;
	astBrakeReleaseTable[udiStepIndex].xEndCMD				:= FALSE;
	
	TPL.FC_LastStep(udiStepIndex, diStep);
	astBrakeReleaseTable[udiStepIndex].sTitle				:= 'End';
	astBrakeReleaseTable[udiStepIndex].udiModuleName		:= 0;
	astBrakeReleaseTable[udiStepIndex].diStep				:= diStep;
	astBrakeReleaseTable[udiStepIndex].diCMD				:= 0;
	astBrakeReleaseTable[udiStepIndex].timTimeOut			:= T#0MS;
	astBrakeReleaseTable[udiStepIndex].xEndCMD				:= TRUE;
	
	TPL.FC_NextCmdTable(iq_udiTableIndex:= udiTableIndex);
	astListofCMDTables[udiTableIndex].sTitle				:= 'Brake Release';
	astListofCMDTables[udiTableIndex].diCMD					:= ET_Cmd.BrakeRelease;
	astListofCMDTables[udiTableIndex].udiNumberOfCmdSteps	:= udiStepIndex;
//
			
// End of system generated code, could be modified for your application -)
END_ACTION

ACTION Init_SubModules:
(* System generated code, could be modified for your application *)

(* Module Group declaration *)

(* aaudiSubModuleGroups[c_udiAlphaGroup1-TPL.Gc_udiGroupOffset,TPL.ET_Group.Member1]	:= c_udiMaster; *)	(* The c_diMaster is the first element of the group c_diAlphaGroup1 *)
(* aaudiSubModuleGroups[c_udiAlphaGroup1-TPL.Gc_udiGroupOffset,TPL.ET_Group.Member2]	:= 0;			*)	(* There is no second element of the group c_diAlphaGroup1 *)

(* aaudiSubModuleGroups[c_udiAlphaGroup2-TPL.Gc_udiGroupOffset,TPL.ET_Group.Member1]	:= 0;			*)	(* There is no first element of the group c_diAlphaGroup2 *)
(* aaudiSubModuleGroups[c_udiAlphaGroup2-TPL.Gc_udiGroupOffset,TPL.ET_Group.Member2]	:= 0;			*)	(* There is no second element of the group c_diAlphaGroup2 *)

(* End of system generated code, could be modified for your application *)


(* System generated code, do not change without consulting 'Schneider Electric Automation GmbH' - otherwise you risk instability!!!*)
xInitSubModulesException := FALSE;

//-------------------------------------------------------------------------------------------------------------------
//-- Set IDs of SubModules *)	
//
	TPL.FC_SetSubModuleIds(	i_udiMainModuleId			:= iq_stStandardModuleItf.i_udiModuleId,
							i_pstSubModulesItf			:= ADR(astSubModuleInterface),
							i_udiNumberOfSubModules		:= c_udiNumberOfSubModules,
							q_etDiag					=> etDiag,
							q_etDiagExt					=> etDiagExtTPL);
						
	IF etDiag <> GD.ET_Diag.Ok AND NOT xInitSubModulesException THEN
		xInitSubModulesException := TRUE;
		
		stInitSubModulesException.sMsg := PDL.FC_MultiConcat(	i_sString1 := 'SetSubModuleIds - ', 
																i_sString2 := GD.FC_EtDiagToString(i_etDiag := etDiag), 
																i_sString3 := ' - ', 
																i_sString4 := TPL.FC_EtDiagExtToString(i_etDiagExt := etDiagExtTPL));
	END_IF	

//-------------------------------------------------------------------------------------------------------------------
//-- Set exception if any exception occurred *)
//
	fbExceptionHandler.SetException(i_xExceptionActive	:= xInitSubModulesException, 
									iq_stException		:= stInitSubModulesException, 
									iq_stExceptionList	:= iq_stExceptionList);
	
	xInitSuccessful := xInitSuccessful AND NOT xInitSubModulesException;
						
	etDiag := GD.ET_Diag.Ok;
//
(* End of system generated code, do not change without consulting 'Schneider Electric Automation GmbH' - otherwise you risk instability!!!*)
END_ACTION

ACTION ExceptionControl_Action:
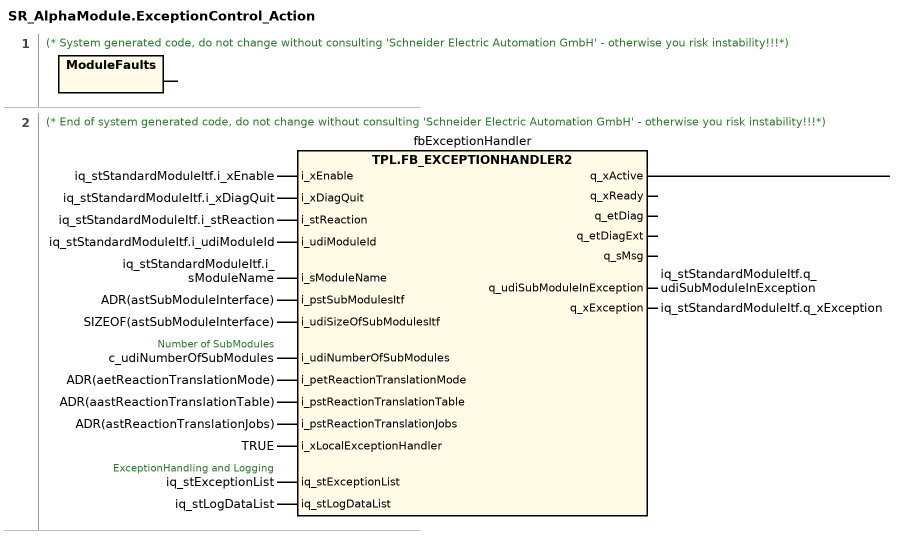
// NETWORK 1
// (* System generated code, do not change without consulting 'Schneider Electric Automation GmbH' - otherwise you risk instability!!!*)
ModuleFaults();

// NETWORK 2
// (* End of system generated code, do not change without consulting 'Schneider Electric Automation GmbH' - otherwise you risk instability!!!*)
//   fbExceptionHandler: ExceptionHandling related variables
//   c_udiNumberOfSubModules: Number of SubModules
//   iq_stExceptionList: ExceptionHandling and Logging
fbExceptionHandler(
    i_xEnable := iq_stStandardModuleItf.i_xEnable,
    i_xDiagQuit := iq_stStandardModuleItf.i_xDiagQuit,
    i_stReaction := iq_stStandardModuleItf.i_stReaction,
    i_udiModuleId := iq_stStandardModuleItf.i_udiModuleId,
    i_sModuleName := iq_stStandardModuleItf.i_sModuleName,
    i_pstSubModulesItf := ADR(astSubModuleInterface),
    i_udiSizeOfSubModulesItf := SIZEOF(astSubModuleInterface),
    i_udiNumberOfSubModules := c_udiNumberOfSubModules,
    i_petReactionTranslationMode := ADR(aetReactionTranslationMode),
    i_pstReactionTranslationTable := ADR(aastReactionTranslationTable),
    i_pstReactionTranslationJobs := ADR(astReactionTranslationJobs),
    i_xLocalExceptionHandler := TRUE,
    iq_stExceptionList := iq_stExceptionList,
    iq_stLogDataList := iq_stLogDataList,
    q_udiSubModuleInException => iq_stStandardModuleItf.q_udiSubModuleInException,
    q_xException => iq_stStandardModuleItf.q_xException); // TPL.FB_EXCEPTIONHANDLER2
END_ACTION

ACTION Init_Exceptions:
(* System generated code, could be modified for your application *)
stUpdateStructsException.etDiag												:= GD.ET_Diag.UnexpectedProgramBehavior;
stUpdateStructsException.udiDiagExt											:= ET_DiagExt.UpdateStructsException;
stUpdateStructsException.sDiagExt											:= FC_EtDiagExtToString(stUpdateStructsException.udiDiagExt);
stUpdateStructsException.sMsg												:= '';	(* Replaced on usage *)
stUpdateStructsException.udiModuleId										:= iq_stStandardModuleItf.i_udiModuleId;
stUpdateStructsException.sModuleName										:= iq_stStandardModuleItf.i_sModuleName;
stUpdateStructsException.stReaction.axReaction[TPL.ET_Reaction.AsyncStop]	:= TRUE;
stUpdateStructsException.etSource											:= TPL.ET_ExceptionSource.NodeModule;
stUpdateStructsException.timDelayTime										:= T#0MS;
stUpdateStructsException.wHmiAttributes										:= 0;
stUpdateStructsException.xAutoQuit											:= FALSE;

stInitReactionsException.etDiag												:= GD.ET_Diag.UnexpectedProgramBehavior;
stInitReactionsException.udiDiagExt											:= ET_DiagExt.InitReactionsException;
stInitReactionsException.sDiagExt											:= FC_EtDiagExtToString(stInitReactionsException.udiDiagExt);
stInitReactionsException.sMsg												:= '';	(* Replaced on usage *)
stInitReactionsException.udiModuleId										:= iq_stStandardModuleItf.i_udiModuleId;
stInitReactionsException.sModuleName										:= iq_stStandardModuleItf.i_sModuleName;
stInitReactionsException.stReaction.axReaction[TPL.ET_Reaction.AsyncStop]	:= TRUE;
stInitReactionsException.etSource											:= TPL.ET_ExceptionSource.NodeModule;
stInitReactionsException.timDelayTime										:= T#0MS;
stInitReactionsException.wHmiAttributes										:= 0;
stInitReactionsException.xAutoQuit											:= FALSE;

